// §3.8b/§3.10.2 — declare one editable value, at Setup. Registration is the ONLY
// thing that makes a value writable; publication, browsability and DATA_WRITE
// never are. All inputs are explicit for TwinCAT 4024 compatibility.
//
// A duplicate key is refused and the FIRST registration stands, because nothing
// here can tell which of the two the author meant. The refusal travels back
// through Setup, where a composition root sees it — rather than an operator
// discovering it later at a control that writes the wrong field.
METHOD M_RegisterConfigWrite : BOOL
VAR_INPUT
    Key           : STRING(160);
    Item          : STRING(255);
    Revision      : UDINT;
    Kind          : E_ConfigKind;
    ValueType     : E_ConfigValueType;
    Storage       : E_ConfigStorage;
    pTarget       : PVOID;
    RequiresReady : BOOL;
    HasMinimum    : BOOL;
    HasMaximum    : BOOL;
    Minimum       : LREAL;
    Maximum       : LREAL;
    Unit          : E_EngUnit;     // NONE = no unit; the HMI shows none
    LabelKey      : STRING(160);
    MaxLength     : UINT;
    EnumDomain    : STRING(255);
    EnumLabelKey  : STRING(80);    // '' = the values are shown as they are
END_VAR
VAR
    i : INT;
END_VAR
M_RegisterConfigWrite := FALSE;
IF _pConfigWrite = 0 THEN _pConfigWrite := ADR(_configWrite); END_IF
IF (Key = '') OR (Revision = 0) OR (pTarget = 0)
OR (Storage = E_ConfigStorage.NONE)
OR (_nConfigWrite >= _configCapacity) THEN
    RETURN;
END_IF
// A text target has a size this code cannot see. Storing 80 characters
// into a STRING(16) would corrupt whatever follows it, so the capacity is
// declared here and the store never exceeds it.
IF (Storage = E_ConfigStorage.AS_STRING)
AND ((MaxLength = 0) OR (MaxLength > 80)) THEN
    RETURN;
END_IF
IF HasMinimum AND HasMaximum AND (Minimum > Maximum) THEN
    RETURN;                                  // an empty range accepts nothing
END_IF
// §3.8e - a line value, and only a line value, is keyed 'line.'. A root publishes
// the line it references under its OWN scope, so the prefix is what keeps the
// line's keys and the root's apart; a mismatch in either direction fails closed.
IF (Kind = E_ConfigKind.LINE_CFG) <> (LEFT(Key, 5) = 'line.') THEN
    RETURN;
END_IF
FOR i := 1 TO _nConfigWrite DO
    IF _pConfigWrite[i - 1].Key = Key THEN
        RETURN;                              // duplicate (Scope, WriteKey): fail closed
    END_IF
END_FOR
_nConfigWrite := _nConfigWrite + 1;
_pConfigWrite[_nConfigWrite - 1].Key := Key;
_pConfigWrite[_nConfigWrite - 1].Item := Item;
_pConfigWrite[_nConfigWrite - 1].Revision := Revision;
_pConfigWrite[_nConfigWrite - 1].Kind := Kind;
_pConfigWrite[_nConfigWrite - 1].ValueType := ValueType;
_pConfigWrite[_nConfigWrite - 1].Storage := Storage;
_pConfigWrite[_nConfigWrite - 1].pTarget := pTarget;
_pConfigWrite[_nConfigWrite - 1].RequiresReady := RequiresReady;
_pConfigWrite[_nConfigWrite - 1].HasMinimum := HasMinimum;
_pConfigWrite[_nConfigWrite - 1].HasMaximum := HasMaximum;
_pConfigWrite[_nConfigWrite - 1].Minimum := Minimum;
_pConfigWrite[_nConfigWrite - 1].Maximum := Maximum;
_pConfigWrite[_nConfigWrite - 1].Unit := Unit;
_pConfigWrite[_nConfigWrite - 1].LabelKey := LabelKey;
_pConfigWrite[_nConfigWrite - 1].MaxLength := MaxLength;
_pConfigWrite[_nConfigWrite - 1].EnumDomain := EnumDomain;
_pConfigWrite[_nConfigWrite - 1].EnumLabelKey := EnumLabelKey;
M_RegisterConfigWrite := TRUE;
END_METHOD

// §3.8c - offer a capture for an ALREADY-REGISTERED editable value. Called at
// Setup, after the M_RegisterConfigWrite that declares the field.
//
// Refused when the key is not registered, which is §3.8c(a) enforced where it
// cannot be bypassed: capture changes how the number arrives, never which
// numbers may change. pSource shall point at a value the module already
// publishes (§3.8c(b)) - the operator has to be able to see the number that is
// about to be stored, on the same screen, before storing it.
METHOD M_RegisterCapture : BOOL
VAR_INPUT
    WriteKey       : STRING(160);
    pSource        : PVOID;
    SourceStorage  : E_ConfigStorage;
END_VAR
VAR
    i : INT;
END_VAR
M_RegisterCapture := FALSE;
IF (WriteKey = '') OR (pSource = 0) OR (SourceStorage = E_ConfigStorage.NONE) THEN
    RETURN;
END_IF
FOR i := 1 TO _nConfigWrite DO
    IF _pConfigWrite[i - 1].Key = WriteKey THEN
        _pConfigWrite[i - 1].pCapture       := pSource;
        _pConfigWrite[i - 1].CaptureStorage := SourceStorage;
        M_RegisterCapture := TRUE;
        RETURN;
    END_IF
END_FOR
END_METHOD

// §3.8c - read the live source as text, so the capture rejoins the ordinary
// write path instead of growing a second typed store. One conversion, one
// validator, one storage routine.
METHOD PRIVATE _M_ReadCaptureText : STRING(255)
VAR_INPUT
    Idx : INT;
END_VAR
VAR
    pB : POINTER TO BOOL;
    pI : POINTER TO INT;
    pD : POINTER TO DINT;
    pU : POINTER TO UDINT;
    pR : POINTER TO REAL;
    pL : POINTER TO LREAL;
    pT : POINTER TO TIME;
    pS : POINTER TO STRING(80);
END_VAR
_M_ReadCaptureText := '';
CASE _pConfigWrite[Idx - 1].CaptureStorage OF
    E_ConfigStorage.AS_BOOL:
        pB := _pConfigWrite[Idx - 1].pCapture;
        _M_ReadCaptureText := SEL(pB^, 'FALSE', 'TRUE');
    E_ConfigStorage.AS_INT:
        pI := _pConfigWrite[Idx - 1].pCapture;
        _M_ReadCaptureText := INT_TO_STRING(pI^);
    E_ConfigStorage.AS_DINT:
        pD := _pConfigWrite[Idx - 1].pCapture;
        _M_ReadCaptureText := DINT_TO_STRING(pD^);
    E_ConfigStorage.AS_UDINT:
        pU := _pConfigWrite[Idx - 1].pCapture;
        _M_ReadCaptureText := UDINT_TO_STRING(pU^);
    E_ConfigStorage.AS_REAL:
        pR := _pConfigWrite[Idx - 1].pCapture;
        _M_ReadCaptureText := REAL_TO_STRING(pR^);
    E_ConfigStorage.AS_LREAL:
        pL := _pConfigWrite[Idx - 1].pCapture;
        _M_ReadCaptureText := LREAL_TO_STRING(pL^);
    E_ConfigStorage.AS_TIME:
        // Whole milliseconds, per the HMI number contract (§3.8b).
        pT := _pConfigWrite[Idx - 1].pCapture;
        _M_ReadCaptureText := DWORD_TO_STRING(TIME_TO_DWORD(pT^));
    E_ConfigStorage.AS_STRING:
        pS := _pConfigWrite[Idx - 1].pCapture;
        _M_ReadCaptureText := pS^;
ELSE
    // Defined ELSE (S5.6): an unset or unknown source class yields empty text,
    // which the write path then refuses to parse. Fail-closed - a capture that
    // cannot read its source stores nothing rather than storing a zero.
    _M_ReadCaptureText := '';
END_CASE
END_METHOD

// §3.8d - put an already-registered value into a data class, and/or raise
// its own minimum levels. Public on purpose: a module TYPE may call it at Setup,
// and so may a composition root that wants a library value in one of the
// PROJECT's classes (a library cannot know a project's classes). The minimums
// only ever raise the class level - see FB_AccessManager.M_DataLevel.
METHOD M_SetConfigAccess : BOOL
VAR_INPUT
    WriteKey      : STRING(160);
    ClassId       : STRING(80);
    MinReadLevel  : E_AccessLevel;
    MinWriteLevel : E_AccessLevel;
END_VAR
VAR
    i : INT;
END_VAR
M_SetConfigAccess := FALSE;
IF (WriteKey = '') OR (LEN(ClassId) > 40)
OR (TO_DINT(MinReadLevel) < TO_DINT(E_AccessLevel.NONE))
OR (TO_DINT(MinReadLevel) > TO_DINT(E_AccessLevel.ADMIN))
OR (TO_DINT(MinWriteLevel) < TO_DINT(E_AccessLevel.NONE))
OR (TO_DINT(MinWriteLevel) > TO_DINT(E_AccessLevel.ADMIN)) THEN
    RETURN;
END_IF
FOR i := 1 TO _nConfigWrite DO
    IF _pConfigWrite[i - 1].Key = WriteKey THEN
        _pConfigWrite[i - 1].ClassId := ClassId;
        _pConfigWrite[i - 1].MinReadLevel := MinReadLevel;
        _pConfigWrite[i - 1].MinWriteLevel := MinWriteLevel;
        M_SetConfigAccess := TRUE;
        RETURN;
    END_IF
END_FOR
END_METHOD

// §3.8d I_ConfigSource - this module's own registry only; composites recurse.
METHOD M_ConfigAccessOf : BOOL
VAR_INPUT
    Scope    : STRING(255);
    WriteKey : STRING(160);
END_VAR
VAR_IN_OUT
    Grant : ST_ConfigAccess;
END_VAR
VAR
    i : INT;
END_VAR
M_ConfigAccessOf := FALSE;
IF (WriteKey = '') OR (Scope <> Status.Name) THEN
    RETURN;
END_IF
FOR i := 1 TO _nConfigWrite DO
    IF _pConfigWrite[i - 1].Key = WriteKey THEN
        Grant.Kind := _pConfigWrite[i - 1].Kind;
        Grant.ClassId := _pConfigWrite[i - 1].ClassId;
        Grant.MinReadLevel := _pConfigWrite[i - 1].MinReadLevel;
        Grant.MinWriteLevel := _pConfigWrite[i - 1].MinWriteLevel;
        M_ConfigAccessOf := TRUE;
        RETURN;
    END_IF
END_FOR
END_METHOD

// §3.8e - TRUE while this module's registered values may not be changed by a
// client: still published, as Writable := FALSE, and refused by the write and
// staging paths. The base is always writable; a line-data MIRROR is not.
METHOD PROTECTED _M_ConfigReadOnly : BOOL
_M_ConfigReadOnly := FALSE;
END_METHOD

// §3.8b — a numeric editable value. Bounds are mandatory here on purpose: an
// unbounded number is the one a client can set to anything, and "what is the
// valid range" is a question the owning module is the only one able to answer.
// Use M_RegisterConfigWrite directly for an unbounded or higher-revision value.
METHOD M_RegisterConfigNumber : BOOL
VAR_INPUT
    Key           : STRING(160);
    Item          : STRING(255);
    LabelKey      : STRING(160);
    Unit          : E_EngUnit;     // every number declares one; NONE = unitless
    Kind          : E_ConfigKind;
    Storage       : E_ConfigStorage;
    pTarget       : PVOID;
    Minimum       : LREAL;
    Maximum       : LREAL;
    RequiresReady : BOOL;
END_VAR
M_RegisterConfigNumber := M_RegisterConfigWrite(Key := Key, Item := Item,
    Revision := 1, Kind := Kind, ValueType := E_ConfigValueType.NUMBER,
    Storage := Storage, pTarget := pTarget, RequiresReady := RequiresReady,
    HasMinimum := TRUE, HasMaximum := TRUE, Minimum := Minimum, Maximum := Maximum,
    Unit := Unit, LabelKey := LabelKey, MaxLength := 0, EnumDomain := '',
    EnumLabelKey := '');
END_METHOD

// §3.8b — an editable TIME, carried and edited as whole milliseconds (the HMI
// validates DURATION as a number; TC3 §3.8 explains the enum spelling).
METHOD M_RegisterConfigDuration : BOOL
VAR_INPUT
    Key           : STRING(160);
    Item          : STRING(255);
    LabelKey      : STRING(160);
    Kind          : E_ConfigKind;
    pTarget       : POINTER TO TIME;
    MinimumMs     : UDINT;
    MaximumMs     : UDINT;
    RequiresReady : BOOL;
END_VAR
M_RegisterConfigDuration := M_RegisterConfigWrite(Key := Key, Item := Item,
    Revision := 1, Kind := Kind, ValueType := E_ConfigValueType.DURATION,
    Storage := E_ConfigStorage.AS_TIME, pTarget := pTarget,
    RequiresReady := RequiresReady, HasMinimum := TRUE, HasMaximum := TRUE,
    Minimum := TO_LREAL(MinimumMs), Maximum := TO_LREAL(MaximumMs),
    Unit := E_EngUnit.MILLISECOND, LabelKey := LabelKey, MaxLength := 0,
    EnumDomain := '', EnumLabelKey := '');
END_METHOD

// §3.8b — an editable BOOL. The exact domain is declared so a client renders a
// choice rather than a free-text field, and so 'yes' is rejected rather than
// silently read as FALSE.
METHOD M_RegisterConfigFlag : BOOL
VAR_INPUT
    Key           : STRING(160);
    Item          : STRING(255);
    LabelKey      : STRING(160);
    Kind          : E_ConfigKind;
    pTarget       : POINTER TO BOOL;
    RequiresReady : BOOL;
END_VAR
M_RegisterConfigFlag := M_RegisterConfigWrite(Key := Key, Item := Item,
    Revision := 1, Kind := Kind, ValueType := E_ConfigValueType.BOOLEAN,
    Storage := E_ConfigStorage.AS_BOOL, pTarget := pTarget,
    RequiresReady := RequiresReady, HasMinimum := FALSE, HasMaximum := FALSE,
    Minimum := 0.0, Maximum := 0.0, Unit := E_EngUnit.NONE, LabelKey := LabelKey,
    MaxLength := 0, EnumDomain := 'TRUE|FALSE', EnumLabelKey := '');
END_METHOD

// §3.8b/§3.10.2 - an editable value that is one of a fixed set, e.g. an
// enumeration stored as its ordinal. Domain lists the exact accepted values
// ('0|1|2'); EnumLabelKey is the catalog prefix the HMI labels each one with
// ('<EnumLabelKey>.<value>'), so a client renders a translated choice and
// anything outside the domain is refused, never read as a default.
METHOD M_RegisterConfigChoice : BOOL
VAR_INPUT
    Key           : STRING(160);
    Item          : STRING(255);
    LabelKey      : STRING(160);
    Kind          : E_ConfigKind;
    Storage       : E_ConfigStorage;
    pTarget       : PVOID;
    Domain        : STRING(255);
    EnumLabelKey  : STRING(80);
    RequiresReady : BOOL;
END_VAR
M_RegisterConfigChoice := FALSE;
IF Domain = '' THEN
    RETURN;                                  // a choice with no choices accepts nothing
END_IF
M_RegisterConfigChoice := M_RegisterConfigWrite(Key := Key, Item := Item,
    Revision := 1, Kind := Kind, ValueType := E_ConfigValueType.NUMBER,
    Storage := Storage, pTarget := pTarget, RequiresReady := RequiresReady,
    HasMinimum := FALSE, HasMaximum := FALSE, Minimum := 0.0, Maximum := 0.0,
    Unit := E_EngUnit.NONE, LabelKey := LabelKey, MaxLength := 0,
    EnumDomain := Domain, EnumLabelKey := EnumLabelKey);
END_METHOD

// §3.8b/§3.10.2 I_ConfigSource — apply one registered write to THIS module.
// The root has already checked DATA_WRITE and subtree ownership; what is left is
// everything only the owner knows. Scope selects the module, so the recursive
// walk asks each module in turn and exactly the one that registered the key
// answers TRUE. An unknown key, a stale revision, or a value the module refuses
// all return FALSE and change nothing.
METHOD M_ApplyConfigWrite : BOOL
VAR_INPUT
    Scope     : STRING(255);
    WriteKey  : STRING(160);
    Revision  : UDINT;
    TextValue : STRING(255);
    RootReady : BOOL;
END_VAR
VAR
    i : INT;
END_VAR
M_ApplyConfigWrite := FALSE;
IF (WriteKey = '') OR (Scope <> Status.Name) OR _M_ConfigReadOnly() THEN
    RETURN;
END_IF
FOR i := 1 TO _nConfigWrite DO
    IF _pConfigWrite[i - 1].Key = WriteKey THEN
        IF _pConfigWrite[i - 1].Revision <> Revision THEN
            RETURN;              // stale capability — the client's metadata is old
        END_IF
        IF _pConfigWrite[i - 1].RequiresReady AND NOT RootReady THEN
            RETURN;
        END_IF
        // The type-specific hook sees the candidate BEFORE anything is stored, so
        // a refusal here is indistinguishable from a range refusal: nothing moved.
        IF NOT _M_OnConfigWrite(WriteKey := WriteKey, TextValue := TextValue) THEN
            RETURN;
        END_IF
        M_ApplyConfigWrite := _M_StoreConfigValue(Idx := i, TextValue := TextValue,
            Commit := TRUE);
        RETURN;
    END_IF
END_FOR
END_METHOD

// §3.8c - apply a capture to THIS module. Resolves the live value and then hands
// it to the ordinary write path, so validation, the type's own invariants, range,
// domain and storage are the SAME code a typed write goes through. A machine-
// supplied number is not more trustworthy than a human-supplied one (§14).
METHOD M_ApplyCapture : BOOL
VAR_INPUT
    Scope     : STRING(255);
    WriteKey  : STRING(160);
    Revision  : UDINT;
    RootReady : BOOL;
END_VAR
VAR
    i : INT;
END_VAR
M_ApplyCapture := FALSE;
IF (WriteKey = '') OR (Scope <> Status.Name) THEN
    RETURN;
END_IF
FOR i := 1 TO _nConfigWrite DO
    IF _pConfigWrite[i - 1].Key = WriteKey THEN
        // No capture registered for this field: refuse rather than fall back to
        // some default, so an unoffered capture can never quietly store a zero.
        IF _pConfigWrite[i - 1].pCapture = 0 THEN
            RETURN;
        END_IF
        M_ApplyCapture := M_ApplyConfigWrite(Scope := Scope, WriteKey := WriteKey,
            Revision := Revision, TextValue := _M_ReadCaptureText(Idx := i),
            RootReady := RootReady);
        RETURN;
    END_IF
END_FOR
END_METHOD

// §3.10.2 — module-specific invariants a generic type/range check cannot state:
// a value that must stay below another, a device that must be idle first. The
// base accepts; the framework still validates revision, type, range and domain
// and stores only after this returns TRUE. Two rules for an override: it shall
// have no side effects, because this runs on a candidate that may still be
// rejected; and it sees the RAW text, not a parsed value — 'abc' reaches it
// exactly as '7' does, so it must never assume the candidate is a number.
METHOD PROTECTED _M_OnConfigWrite : BOOL
VAR_INPUT
    WriteKey  : STRING(160);
    TextValue : STRING(255);
END_VAR
_M_OnConfigWrite := TRUE;
END_METHOD

// §3.8b/§5.6 — validate a candidate completely, then store it. Every rejection
// happens before the first byte moves, so a refused write leaves the module
// exactly as it was. Range is checked against BOTH the declared bounds and the
// storage type's own limits: a DINT field with no declared maximum still cannot
// be handed 1E30.
//
// Commit := FALSE runs the IDENTICAL validation and stores nothing. That is the
// staging pass of a §3.8b set load, and it deliberately shares this code rather
// than restating the rules: a validator that can disagree with the writer is
// worse than no validator, because it makes an all-or-nothing load claim an
// atomicity it does not have.
METHOD PROTECTED _M_StoreConfigValue : BOOL
VAR_INPUT
    Idx       : INT;
    TextValue : STRING(255);
    Commit    : BOOL;
END_VAR
VAR
    num : LREAL;
    pB  : POINTER TO BOOL;
    pI  : POINTER TO INT;
    pD  : POINTER TO DINT;
    pU  : POINTER TO UDINT;
    pR  : POINTER TO REAL;
    pL  : POINTER TO LREAL;
    pT  : POINTER TO TIME;
    pS  : POINTER TO STRING(80);
END_VAR
_M_StoreConfigValue := FALSE;
IF (Idx < 1) OR (Idx > _nConfigWrite) OR (_pConfigWrite[Idx - 1].pTarget = 0) THEN
    RETURN;
END_IF
// A declared domain is exact and is checked on the raw text, whatever the type.
IF _pConfigWrite[Idx - 1].EnumDomain <> '' THEN
    IF NOT _M_InEnumDomain(Domain := _pConfigWrite[Idx - 1].EnumDomain,
            Text := TextValue) THEN
        RETURN;
    END_IF
END_IF
IF _pConfigWrite[Idx - 1].Storage = E_ConfigStorage.AS_BOOL THEN
    pB := _M_Target(Idx := Idx);
    IF (TextValue = 'TRUE') OR (TextValue = 'true') OR (TextValue = 'True')
    OR (TextValue = '1') THEN
        IF Commit THEN
            pB^ := TRUE;
        END_IF
    ELSIF (TextValue = 'FALSE') OR (TextValue = 'false') OR (TextValue = 'False')
    OR (TextValue = '0') THEN
        IF Commit THEN
            pB^ := FALSE;
        END_IF
    ELSE
        RETURN;
    END_IF
    _M_StoreConfigValue := TRUE;
    RETURN;
END_IF
IF _pConfigWrite[Idx - 1].Storage = E_ConfigStorage.AS_STRING THEN
    IF TO_UINT(LEN(TextValue)) > _pConfigWrite[Idx - 1].MaxLength THEN
        RETURN;                              // would truncate: reject, never trim
    END_IF
    IF Commit THEN
        pS := _M_Target(Idx := Idx);
        pS^ := TextValue;
    END_IF
    _M_StoreConfigValue := TRUE;
    RETURN;
END_IF
// Everything else is numeric.
IF NOT F_TryParseNumber(Text := TextValue, Value => num) THEN
    RETURN;
END_IF
IF _pConfigWrite[Idx - 1].HasMinimum AND (num < _pConfigWrite[Idx - 1].Minimum) THEN
    RETURN;
END_IF
IF _pConfigWrite[Idx - 1].HasMaximum AND (num > _pConfigWrite[Idx - 1].Maximum) THEN
    RETURN;
END_IF
CASE _pConfigWrite[Idx - 1].Storage OF
    E_ConfigStorage.AS_INT:
        IF (num < -32768.0) OR (num > 32767.0) THEN
            RETURN;
        END_IF
        // Two statements, not one condition: IEC 61131-3 does not mandate
        // short-circuit evaluation and TwinCAT's option for it is off by
        // default, so a combined test would still convert a value the range
        // check is there to reject (§5.6).
        IF num <> TO_LREAL(TO_LINT(num)) THEN
            RETURN;
        END_IF
        IF Commit THEN
            pI := _M_Target(Idx := Idx);
            pI^ := LREAL_TO_INT(num);
        END_IF
    E_ConfigStorage.AS_DINT:
        IF (num < -2147483648.0) OR (num > 2147483647.0) THEN
            RETURN;
        END_IF
        IF num <> TO_LREAL(TO_LINT(num)) THEN
            RETURN;
        END_IF
        IF Commit THEN
            pD := _M_Target(Idx := Idx);
            pD^ := LREAL_TO_DINT(num);
        END_IF
    E_ConfigStorage.AS_UDINT:
        IF (num < 0.0) OR (num > 4294967295.0) THEN
            RETURN;
        END_IF
        IF num <> TO_LREAL(TO_LINT(num)) THEN
            RETURN;
        END_IF
        IF Commit THEN
            pU := _M_Target(Idx := Idx);
            pU^ := LREAL_TO_UDINT(num);
        END_IF
    E_ConfigStorage.AS_REAL:
        IF (num < -3.402823E38) OR (num > 3.402823E38) THEN
            RETURN;
        END_IF
        IF Commit THEN
            pR := _M_Target(Idx := Idx);
            pR^ := LREAL_TO_REAL(num);
        END_IF
    E_ConfigStorage.AS_LREAL:
        IF Commit THEN
            pL := _M_Target(Idx := Idx);
            pL^ := num;
        END_IF
    E_ConfigStorage.AS_TIME:
        // Whole milliseconds: a duration is not a place for a rounding surprise.
        IF (num < 0.0) OR (num > 4294967295.0) THEN
            RETURN;
        END_IF
        IF num <> TO_LREAL(TO_LINT(num)) THEN
            RETURN;
        END_IF
        IF Commit THEN
            pT := _M_Target(Idx := Idx);
            pT^ := UDINT_TO_TIME(LREAL_TO_UDINT(num));
        END_IF
ELSE
    RETURN;
END_CASE
_M_StoreConfigValue := TRUE;
END_METHOD

// §3.10.2 — the current value of a registered entry, in the serialization the
// client validates and writes back. Read live from the target every walk: a
// cached copy would let the manifest disagree with the machine.
METHOD PROTECTED _M_ConfigValueText : STRING(255)
VAR_INPUT
    Idx : INT;
END_VAR
VAR
    pB : POINTER TO BOOL;
    pI : POINTER TO INT;
    pD : POINTER TO DINT;
    pU : POINTER TO UDINT;
    pR : POINTER TO REAL;
    pL : POINTER TO LREAL;
    pT : POINTER TO TIME;
    pS : POINTER TO STRING(80);
END_VAR
_M_ConfigValueText := '';
IF (Idx < 1) OR (Idx > _nConfigWrite) OR (_pConfigWrite[Idx - 1].pTarget = 0) THEN
    RETURN;
END_IF
CASE _pConfigWrite[Idx - 1].Storage OF
    E_ConfigStorage.AS_BOOL:
        pB := _M_Target(Idx := Idx);
        IF pB^ THEN
            _M_ConfigValueText := 'TRUE';
        ELSE
            _M_ConfigValueText := 'FALSE';
        END_IF
    E_ConfigStorage.AS_INT:
        pI := _M_Target(Idx := Idx);
        _M_ConfigValueText := TO_STRING(pI^);
    E_ConfigStorage.AS_DINT:
        pD := _M_Target(Idx := Idx);
        _M_ConfigValueText := TO_STRING(pD^);
    E_ConfigStorage.AS_UDINT:
        pU := _M_Target(Idx := Idx);
        _M_ConfigValueText := TO_STRING(pU^);
    E_ConfigStorage.AS_REAL:
        pR := _M_Target(Idx := Idx);
        _M_ConfigValueText := TO_STRING(pR^);
    E_ConfigStorage.AS_LREAL:
        pL := _M_Target(Idx := Idx);
        _M_ConfigValueText := TO_STRING(pL^);
    E_ConfigStorage.AS_TIME:
        pT := _M_Target(Idx := Idx);
        _M_ConfigValueText := TO_STRING(TIME_TO_UDINT(pT^));
    E_ConfigStorage.AS_STRING:
        pS := _M_Target(Idx := Idx);
        _M_ConfigValueText := pS^;
END_CASE
END_METHOD

// §3.10.2 — exact membership in a pipe-separated domain. Exact means exact: no
// trimming, no case folding. The client was given this list and can send one of
// its entries.
METHOD PRIVATE _M_InEnumDomain : BOOL
VAR_INPUT
    Domain : STRING(255);
    Text   : STRING(255);
END_VAR
VAR
    rest  : STRING(255);
    token : STRING(255);
    pos   : INT;
    i     : INT;
END_VAR
_M_InEnumDomain := FALSE;
rest := Domain;
FOR i := 1 TO 32 DO                          // bounded scan (§5.6)
    IF rest = '' THEN
        RETURN;
    END_IF
    pos := FIND(rest, '|');
    IF pos = 0 THEN
        token := rest;
        rest := '';
    ELSE
        token := LEFT(rest, pos - 1);
        rest := MID(rest, TO_INT(LEN(rest)) - pos, pos + 1);
    END_IF
    IF token = Text THEN
        _M_InEnumDomain := TRUE;
        RETURN;
    END_IF
END_FOR
END_METHOD

// §3.8b I_ConfigSource — would this write be accepted? Byte-for-byte the
// lookup and gating of M_ApplyConfigWrite, then the shared validator with
// Commit := FALSE. Nothing in this module changes, including through the
// type-specific invariant hook, which §3.10.2 already requires to be free of
// side effects because it runs on a candidate that may still be rejected.
METHOD M_StageConfigWrite : BOOL
VAR_INPUT
    Scope     : STRING(255);
    WriteKey  : STRING(160);
    Revision  : UDINT;
    TextValue : STRING(255);
    RootReady : BOOL;
END_VAR
VAR
    i : INT;
END_VAR
M_StageConfigWrite := FALSE;
IF (WriteKey = '') OR (Scope <> Status.Name) OR _M_ConfigReadOnly() THEN
    RETURN;
END_IF
FOR i := 1 TO _nConfigWrite DO
    IF _pConfigWrite[i - 1].Key = WriteKey THEN
        IF _pConfigWrite[i - 1].Revision <> Revision THEN
            RETURN;
        END_IF
        IF _pConfigWrite[i - 1].RequiresReady AND NOT RootReady THEN
            RETURN;
        END_IF
        IF NOT _M_OnConfigWrite(WriteKey := WriteKey, TextValue := TextValue) THEN
            RETURN;
        END_IF
        M_StageConfigWrite := _M_StoreConfigValue(Idx := i, TextValue := TextValue,
            Commit := FALSE);
        RETURN;
    END_IF
END_FOR
END_METHOD

// §3.8b — the restore rule for one retained StationCfg image, written ONCE here
// so no module type carries its own copy of it (§1.1 O1).
//
// Every StationCfg structure shall carry SchemaVersion : UINT as its FIRST
// member, and this decides what a given value of it means:
//
//   version = SchemaVersion  -> restored. Returns TRUE; the caller keeps the
//                               retained values and does nothing.
//   version = 0              -> never written. A first boot has lost nothing,
//                               so it initializes SILENTLY: returns FALSE with
//                               no annunciation, and the caller writes defaults.
//   anything else            -> a REAL image was rejected. Returns FALSE and
//                               records the loss for the root to annunciate with
//                               this module's canonical path.
//
// The version is stamped forward either way, so the next boot is an ordinary
// restore rather than a repeated annunciation. What is NOT done is reading the
// unrecognized image by field position: that is precisely how a changed layout
// becomes a plausible wrong number instead of an honest default.
//
// The consequence of a loss belongs to the deployment, not to this module —
// E_ConfigRestorePolicy at the root decides whether the station runs and
// annunciates or refuses START_STOP until an ENGINEER acknowledges. A module
// that faulted itself here would take that decision away from the deployment.
METHOD M_RestoreStationCfg : BOOL
VAR_INPUT
    pVersion      : POINTER TO UINT;   // ADR of the structure's FIRST member
    SchemaVersion : UINT;              // the layout this build understands
END_VAR
M_RestoreStationCfg := FALSE;
IF pVersion = 0 THEN
    RETURN;                              // unwired: defaults, and never a claim
END_IF
IF SchemaVersion = 0 THEN
    RETURN;                              // 0 is reserved for "never written"
END_IF
IF pVersion^ = SchemaVersion THEN
    M_RestoreStationCfg := TRUE;
    RETURN;
END_IF
IF pVersion^ <> 0 THEN
    // A real image was rejected. The station will run on defaults and it will
    // say so — the difference between an empty machine and one that has just
    // lost its commissioning is exactly what an operator needs told.
    _restoreLost := TRUE;
    _restoreFound := pVersion^;
    _restoreExpected := SchemaVersion;
END_IF
pVersion^ := SchemaVersion;
END_METHOD

// §3.8b I_ConfigSource — hand the root this module's unreported restore loss,
// exactly once. Taking it clears the slot, so the root can drain the whole
// subtree in a loop and each loss is annunciated one time per boot.
METHOD M_TakeRestoreLoss : BOOL
VAR_OUTPUT
    Path     : STRING(80);
    Expected : UINT;
    Found    : UINT;
END_VAR
M_TakeRestoreLoss := FALSE;
Path := '';
Expected := 0;
Found := 0;
IF NOT _restoreLost THEN
    RETURN;
END_IF
_restoreLost := FALSE;
Path := Status.Name;
Expected := _restoreExpected;
Found := _restoreFound;
M_TakeRestoreLoss := TRUE;
END_METHOD

// §7.6.1 I_ManualTarget - answer for THIS module only. Same shape as
// M_ApplyConfigWrite: the walk asks every module and exactly the one whose
// Scope matches replies, so routing is a property of registration rather than
// of a chain somebody maintains by hand.
METHOD M_ApplyManual : BOOL
VAR_INPUT
    Scope : STRING(255);
    Value : DINT;
END_VAR
M_ApplyManual := FALSE;
IF Scope <> Status.Name THEN
    RETURN;
END_IF
// ManualCommand still validates the value against the published catalogue and
// still runs the §6.1 lifecycle. Reaching the module is all this adds.
M_ApplyManual := ManualCommand(Value := Value);
END_METHOD

// §7.6.1a I_ManualTarget - the held-command twin of M_ApplyManual. A type with
// no held commands inherits RequestHeldCommand's refusal, so an unsupported
// hold is a defined FALSE.
METHOD M_ApplyHeld : BOOL
VAR_INPUT
    Scope  : STRING(255);
    Value  : DINT;
    Enable : ST_ManualEnableStatus;
END_VAR
M_ApplyHeld := FALSE;
IF Scope <> Status.Name THEN
    RETURN;
END_IF
M_ApplyHeld := RequestHeldCommand(Value := Value, Enable := Enable);
END_METHOD

// Optional owner storage selected before any registration; base modules keep twelve slots.
METHOD PROTECTED _M_UseConfigRegistry : BOOL
VAR_INPUT
    pRecords : POINTER TO ST_ConfigWriteDef;
    Capacity : INT;
END_VAR
_M_UseConfigRegistry := FALSE;
IF (_nConfigWrite <> 0) OR (pRecords = 0) OR (Capacity < 1)
OR (Capacity > PL_Fraktal.MAX_LINE_RECORDS) THEN RETURN; END_IF
_pConfigWrite := pRecords;
_configCapacity := Capacity;
_M_UseConfigRegistry := TRUE;
END_METHOD

END_FUNCTION_BLOCK

// ---- Platform/F_RationalizeDiagnostic.TcPOU
// Core §8.9 — apply the one generated priority/category to a diagnostic at its
// source. Unknown external reasons keep the caller values until their owning
// AlarmLog joins a validated runtime record.
FUNCTION F_RationalizeDiagnostic : BOOL
VAR_IN_OUT
    Diag : ST_Diagnostic;
END_VAR
VAR
    meta : ST_AlarmMeta;
END_VAR

F_RationalizeDiagnostic := F_ReasonMeta(
    Reason := Diag.ReasonCode, Meta := meta);
IF F_RationalizeDiagnostic THEN
    Diag.Severity := meta.Priority;
    Diag.Category := meta.Category;
END_IF

END_FUNCTION

// ---- Platform/F_ReasonMeta.TcPOU
// Core §8.9 — resolve one generated rationalization by ReasonCode.
FUNCTION F_ReasonMeta : BOOL
VAR_INPUT
    Reason : E_Reason;
END_VAR
VAR_IN_OUT
    Meta : ST_AlarmMeta;
END_VAR
VAR
    i : INT;
    candidate : ST_AlarmMeta;
END_VAR

F_ReasonMeta := FALSE;
FOR i := 1 TO PL_ReasonCatalog.COUNT DO
    IF F_ReasonMetaByIndex(Index := i, Meta := candidate)
    AND (candidate.ReasonCode = Reason) THEN
        Meta := candidate;
        F_ReasonMeta := TRUE;
        RETURN;
    END_IF
END_FOR

END_FUNCTION

// ---- Platform/F_ReasonMetaByIndex.TcPOU
// GENERATED FILE — DO NOT EDIT. Core §8.8/§8.9 complete catalog projection.
FUNCTION F_ReasonMetaByIndex : BOOL
VAR_INPUT
    Index : INT;
END_VAR
VAR_IN_OUT
    Meta : ST_AlarmMeta;
END_VAR

F_ReasonMetaByIndex := FALSE;
Meta.ReasonCode := E_Reason.NONE;
Meta.OperatorAction := '';
Meta.Consequence := '';
Meta.Priority := E_Severity.LOW;
Meta.Category := E_Category.PROCESS;
Meta.Shelvable := FALSE;
CASE Index OF
    1:
        Meta.ReasonCode := 10;
        Meta.OperatorAction := 'std.reason.10.action';
        Meta.Consequence := 'std.reason.10.consequence';
        Meta.Priority := E_Severity.MED;
        Meta.Category := E_Category.SYSTEM;
        Meta.Shelvable := FALSE;
    2:
        Meta.ReasonCode := 11;
        Meta.OperatorAction := 'std.reason.11.action';
        Meta.Consequence := 'std.reason.11.consequence';
        Meta.Priority := E_Severity.LOW;
        Meta.Category := E_Category.SYSTEM;
        Meta.Shelvable := TRUE;
    3:
        Meta.ReasonCode := 12;
        Meta.OperatorAction := 'std.reason.12.action';
        Meta.Consequence := 'std.reason.12.consequence';
        Meta.Priority := E_Severity.LOW;
        Meta.Category := E_Category.SYSTEM;
        Meta.Shelvable := TRUE;
    4:
        Meta.ReasonCode := 13;
        Meta.OperatorAction := 'std.reason.13.action';
        Meta.Consequence := 'std.reason.13.consequence';
        Meta.Priority := E_Severity.MED;
        Meta.Category := E_Category.SYSTEM;
        Meta.Shelvable := FALSE;
    5:
        Meta.ReasonCode := 14;
        Meta.OperatorAction := 'std.reason.14.action';
        Meta.Consequence := 'std.reason.14.consequence';
        Meta.Priority := E_Severity.MED;
        Meta.Category := E_Category.SYSTEM;
        Meta.Shelvable := FALSE;
    6:
        Meta.ReasonCode := 15;
        Meta.OperatorAction := 'std.reason.15.action';
        Meta.Consequence := 'std.reason.15.consequence';
        Meta.Priority := E_Severity.HIGH;
        Meta.Category := E_Category.SYSTEM;
        Meta.Shelvable := FALSE;
    7:
        Meta.ReasonCode := 16;
        Meta.OperatorAction := 'std.reason.16.action';
        Meta.Consequence := 'std.reason.16.consequence';
        Meta.Priority := E_Severity.LOW;
        Meta.Category := E_Category.SYSTEM;
        Meta.Shelvable := TRUE;
    8:
        Meta.ReasonCode := 17;
        Meta.OperatorAction := 'std.reason.17.action';
        Meta.Consequence := 'std.reason.17.consequence';
        Meta.Priority := E_Severity.LOW;
        Meta.Category := E_Category.SYSTEM;
        Meta.Shelvable := TRUE;
    9:
        Meta.ReasonCode := 18;
        Meta.OperatorAction := 'std.reason.18.action';
        Meta.Consequence := 'std.reason.18.consequence';
        Meta.Priority := E_Severity.MED;
        Meta.Category := E_Category.SYSTEM;
        Meta.Shelvable := FALSE;
    10:
        Meta.ReasonCode := 19;
        Meta.OperatorAction := 'std.reason.19.action';
        Meta.Consequence := 'std.reason.19.consequence';
        Meta.Priority := E_Severity.LOW;
        Meta.Category := E_Category.SYSTEM;
        Meta.Shelvable := TRUE;
    11:
        Meta.ReasonCode := 20;
        Meta.OperatorAction := 'std.reason.20.action';
        Meta.Consequence := 'std.reason.20.consequence';
        Meta.Priority := E_Severity.MED;
        Meta.Category := E_Category.SYSTEM;
        Meta.Shelvable := FALSE;
    12:
        Meta.ReasonCode := 21;
        Meta.OperatorAction := 'std.reason.21.action';
        Meta.Consequence := 'std.reason.21.consequence';
        Meta.Priority := E_Severity.LOW;
        Meta.Category := E_Category.SYSTEM;
        Meta.Shelvable := TRUE;
    13:
        Meta.ReasonCode := 2001;
        Meta.OperatorAction := 'std.reason.2001.action';
        Meta.Consequence := 'std.reason.2001.consequence';
        Meta.Priority := E_Severity.MED;
        Meta.Category := E_Category.PROCESS;
        Meta.Shelvable := FALSE;
    14:
        Meta.ReasonCode := 2002;
        Meta.OperatorAction := 'std.reason.2002.action';
        Meta.Consequence := 'std.reason.2002.consequence';
        Meta.Priority := E_Severity.LOW;
        Meta.Category := E_Category.PROCESS;
        Meta.Shelvable := FALSE;
    15:
        Meta.ReasonCode := 2003;
        Meta.OperatorAction := 'std.reason.2003.action';
        Meta.Consequence := 'std.reason.2003.consequence';
        Meta.Priority := E_Severity.MED;
        Meta.Category := E_Category.PROCESS;
        Meta.Shelvable := FALSE;
    16:
        Meta.ReasonCode := 2004;
        Meta.OperatorAction := 'std.reason.2004.action';
        Meta.Consequence := 'std.reason.2004.consequence';
        Meta.Priority := E_Severity.MED;
        Meta.Category := E_Category.PROCESS;
        Meta.Shelvable := FALSE;
    17:
        Meta.ReasonCode := 2005;
        Meta.OperatorAction := 'std.reason.2005.action';
        Meta.Consequence := 'std.reason.2005.consequence';
        Meta.Priority := E_Severity.LOW;
        Meta.Category := E_Category.PROCESS;
        Meta.Shelvable := TRUE;
    18:
        Meta.ReasonCode := 2006;
        Meta.OperatorAction := 'std.reason.2006.action';
        Meta.Consequence := 'std.reason.2006.consequence';
        Meta.Priority := E_Severity.MED;
        Meta.Category := E_Category.PROCESS;
        Meta.Shelvable := FALSE;
    19:
        Meta.ReasonCode := 2007;
        Meta.OperatorAction := 'std.reason.2007.action';
        Meta.Consequence := 'std.reason.2007.consequence';
        Meta.Priority := E_Severity.LOW;
        Meta.Category := E_Category.PROCESS;
        Meta.Shelvable := TRUE;
    20:
        Meta.ReasonCode := 2008;
        Meta.OperatorAction := 'std.reason.2008.action';
        Meta.Consequence := 'std.reason.2008.consequence';
        Meta.Priority := E_Severity.LOW;
        Meta.Category := E_Category.PROCESS;
        Meta.Shelvable := FALSE;
    21:
        Meta.ReasonCode := 2010;
        Meta.OperatorAction := 'std.reason.2010.action';
        Meta.Consequence := 'std.reason.2010.consequence';
        Meta.Priority := E_Severity.MED;
        Meta.Category := E_Category.SYSTEM;
        Meta.Shelvable := FALSE;
    22:
        Meta.ReasonCode := 2011;
        Meta.OperatorAction := 'std.reason.2011.action';
        Meta.Consequence := 'std.reason.2011.consequence';
        Meta.Priority := E_Severity.LOW;
        Meta.Category := E_Category.PROCESS;
        Meta.Shelvable := TRUE;
    23:
        Meta.ReasonCode := 2012;
        Meta.OperatorAction := 'std.reason.2012.action';
        Meta.Consequence := 'std.reason.2012.consequence';
        Meta.Priority := E_Severity.MED;
        Meta.Category := E_Category.SYSTEM;
        Meta.Shelvable := FALSE;
    24:
        Meta.ReasonCode := 2020;
        Meta.OperatorAction := 'std.reason.2020.action';
        Meta.Consequence := 'std.reason.2020.consequence';
        Meta.Priority := E_Severity.MED;
        Meta.Category := E_Category.SYSTEM;
        Meta.Shelvable := FALSE;
    25:
        Meta.ReasonCode := 2021;
        Meta.OperatorAction := 'std.reason.2021.action';
        Meta.Consequence := 'std.reason.2021.consequence';
        Meta.Priority := E_Severity.MED;
        Meta.Category := E_Category.SYSTEM;
        Meta.Shelvable := FALSE;
    26:
        Meta.ReasonCode := 2022;
        Meta.OperatorAction := 'std.reason.2022.action';
        Meta.Consequence := 'std.reason.2022.consequence';
        Meta.Priority := E_Severity.HIGH;
        Meta.Category := E_Category.PROCESS;
        Meta.Shelvable := FALSE;
    27:
        Meta.ReasonCode := 2023;
        Meta.OperatorAction := 'std.reason.2023.action';
        Meta.Consequence := 'std.reason.2023.consequence';
        Meta.Priority := E_Severity.MED;
        Meta.Category := E_Category.PROCESS;
        Meta.Shelvable := FALSE;
    28:
        Meta.ReasonCode := 2024;
        Meta.OperatorAction := '';
        Meta.Consequence := 'std.reason.2024.consequence';
        Meta.Priority := E_Severity.LOW;
        Meta.Category := E_Category.PROCESS;
        Meta.Shelvable := FALSE;
    29:
        Meta.ReasonCode := 2025;
        Meta.OperatorAction := '';
        Meta.Consequence := 'std.reason.2025.consequence';
        Meta.Priority := E_Severity.LOW;
        Meta.Category := E_Category.PROCESS;
        Meta.Shelvable := FALSE;
    30:
        Meta.ReasonCode := 2026;
        Meta.OperatorAction := '';
        Meta.Consequence := 'std.reason.2026.consequence';
        Meta.Priority := E_Severity.LOW;
        Meta.Category := E_Category.PROCESS;
        Meta.Shelvable := FALSE;
    31:
        Meta.ReasonCode := 2027;
        Meta.OperatorAction := '';
        Meta.Consequence := 'std.reason.2027.consequence';
        Meta.Priority := E_Severity.LOW;
        Meta.Category := E_Category.PROCESS;
        Meta.Shelvable := FALSE;
    32:
        Meta.ReasonCode := 2030;
        Meta.OperatorAction := 'std.reason.2030.action';
        Meta.Consequence := 'std.reason.2030.consequence';
        Meta.Priority := E_Severity.LOW;
        Meta.Category := E_Category.SYSTEM;
        Meta.Shelvable := FALSE;
    33:
        Meta.ReasonCode := 2040;
        Meta.OperatorAction := 'std.reason.2040.action';
        Meta.Consequence := 'std.reason.2040.consequence';
        Meta.Priority := E_Severity.MED;
        Meta.Category := E_Category.SYSTEM;
        Meta.Shelvable := FALSE;
    34:
        Meta.ReasonCode := 2041;
        Meta.OperatorAction := 'std.reason.2041.action';
        Meta.Consequence := 'std.reason.2041.consequence';
        Meta.Priority := E_Severity.MED;
        Meta.Category := E_Category.SYSTEM;
        Meta.Shelvable := FALSE;
    35:
        Meta.ReasonCode := 2042;
        Meta.OperatorAction := 'std.reason.2042.action';
        Meta.Consequence := 'std.reason.2042.consequence';
        Meta.Priority := E_Severity.LOW;
        Meta.Category := E_Category.SYSTEM;
        Meta.Shelvable := FALSE;
    36:
        Meta.ReasonCode := 2043;
        Meta.OperatorAction := '';
        Meta.Consequence := 'std.reason.2043.consequence';
        Meta.Priority := E_Severity.LOW;
        Meta.Category := E_Category.SYSTEM;
        Meta.Shelvable := FALSE;
    37:
        Meta.ReasonCode := 2901;
        Meta.OperatorAction := '';
        Meta.Consequence := 'std.reason.2901.consequence';
        Meta.Priority := E_Severity.LOW;
        Meta.Category := E_Category.SYSTEM;
        Meta.Shelvable := FALSE;
    38:
        Meta.ReasonCode := 10001;
        Meta.OperatorAction := 'std.reason.10001.action';
        Meta.Consequence := 'std.reason.10001.consequence';
        Meta.Priority := E_Severity.MED;
        Meta.Category := E_Category.PROCESS;
        Meta.Shelvable := FALSE;
    39:
        Meta.ReasonCode := 10002;
        Meta.OperatorAction := 'std.reason.10002.action';
        Meta.Consequence := 'std.reason.10002.consequence';
        Meta.Priority := E_Severity.MED;
        Meta.Category := E_Category.PROCESS;
        Meta.Shelvable := FALSE;
    40:
        Meta.ReasonCode := 10003;
        Meta.OperatorAction := 'std.reason.10003.action';
        Meta.Consequence := 'std.reason.10003.consequence';
        Meta.Priority := E_Severity.MED;
        Meta.Category := E_Category.PROCESS;
        Meta.Shelvable := FALSE;
    41:
        Meta.ReasonCode := 10004;
        Meta.OperatorAction := 'std.reason.10004.action';
        Meta.Consequence := 'std.reason.10004.consequence';
        Meta.Priority := E_Severity.MED;
        Meta.Category := E_Category.PROCESS;
        Meta.Shelvable := FALSE;
    42:
        Meta.ReasonCode := 10005;
        Meta.OperatorAction := 'std.reason.10005.action';
        Meta.Consequence := 'std.reason.10005.consequence';
        Meta.Priority := E_Severity.MED;
        Meta.Category := E_Category.PROCESS;
        Meta.Shelvable := FALSE;
    43:
        Meta.ReasonCode := 10101;
        Meta.OperatorAction := 'std.reason.10101.action';
        Meta.Consequence := 'std.reason.10101.consequence';
        Meta.Priority := E_Severity.MED;
        Meta.Category := E_Category.PROCESS;
        Meta.Shelvable := FALSE;
    44:
        Meta.ReasonCode := 10102;
        Meta.OperatorAction := 'std.reason.10102.action';
        Meta.Consequence := 'std.reason.10102.consequence';
        Meta.Priority := E_Severity.MED;
        Meta.Category := E_Category.PROCESS;
        Meta.Shelvable := FALSE;
    45:
        Meta.ReasonCode := 10103;
        Meta.OperatorAction := 'std.reason.10103.action';
        Meta.Consequence := 'std.reason.10103.consequence';
        Meta.Priority := E_Severity.HIGH;
        Meta.Category := E_Category.PROCESS;
        Meta.Shelvable := FALSE;
    46:
        Meta.ReasonCode := 10111;
        Meta.OperatorAction := 'std.reason.10111.action';
        Meta.Consequence := 'std.reason.10111.consequence';
        Meta.Priority := E_Severity.MED;
        Meta.Category := E_Category.PROCESS;
        Meta.Shelvable := FALSE;
    47:
        Meta.ReasonCode := 10112;
        Meta.OperatorAction := 'std.reason.10112.action';
        Meta.Consequence := 'std.reason.10112.consequence';
        Meta.Priority := E_Severity.MED;
        Meta.Category := E_Category.PROCESS;
        Meta.Shelvable := FALSE;
    48:
        Meta.ReasonCode := 10113;
        Meta.OperatorAction := 'std.reason.10113.action';
        Meta.Consequence := 'std.reason.10113.consequence';
        Meta.Priority := E_Severity.HIGH;
        Meta.Category := E_Category.PROCESS;
        Meta.Shelvable := FALSE;
    49:
        Meta.ReasonCode := 10114;
        Meta.OperatorAction := 'std.reason.10114.action';
        Meta.Consequence := 'std.reason.10114.consequence';
        Meta.Priority := E_Severity.MED;
        Meta.Category := E_Category.PROCESS;
        Meta.Shelvable := FALSE;
    50:
        Meta.ReasonCode := 10115;
        Meta.OperatorAction := 'std.reason.10115.action';
        Meta.Consequence := 'std.reason.10115.consequence';
        Meta.Priority := E_Severity.MED;
        Meta.Category := E_Category.SYSTEM;
        Meta.Shelvable := FALSE;
    51:
        Meta.ReasonCode := 10116;
        Meta.OperatorAction := 'std.reason.10116.action';
        Meta.Consequence := 'std.reason.10116.consequence';
        Meta.Priority := E_Severity.MED;
        Meta.Category := E_Category.PROCESS;
        Meta.Shelvable := FALSE;
    52:
        Meta.ReasonCode := 10201;
        Meta.OperatorAction := 'std.reason.10201.action';
        Meta.Consequence := 'std.reason.10201.consequence';
        Meta.Priority := E_Severity.MED;
        Meta.Category := E_Category.PROCESS;
        Meta.Shelvable := FALSE;
    53:
        Meta.ReasonCode := 10202;
        Meta.OperatorAction := 'std.reason.10202.action';
        Meta.Consequence := 'std.reason.10202.consequence';
        Meta.Priority := E_Severity.MED;
        Meta.Category := E_Category.PROCESS;
        Meta.Shelvable := FALSE;
    54:
        Meta.ReasonCode := 10203;
        Meta.OperatorAction := 'std.reason.10203.action';
        Meta.Consequence := 'std.reason.10203.consequence';
        Meta.Priority := E_Severity.HIGH;
        Meta.Category := E_Category.SYSTEM;
        Meta.Shelvable := FALSE;
    55:
        Meta.ReasonCode := 10204;
        Meta.OperatorAction := 'std.reason.10204.action';
        Meta.Consequence := 'std.reason.10204.consequence';
        Meta.Priority := E_Severity.MED;
        Meta.Category := E_Category.PROCESS;
        Meta.Shelvable := FALSE;
    56:
        Meta.ReasonCode := 10205;
        Meta.OperatorAction := 'std.reason.10205.action';
        Meta.Consequence := 'std.reason.10205.consequence';
        Meta.Priority := E_Severity.MED;
        Meta.Category := E_Category.PROCESS;
        Meta.Shelvable := FALSE;
    57:
        Meta.ReasonCode := 10206;
        Meta.OperatorAction := 'std.reason.10206.action';
        Meta.Consequence := 'std.reason.10206.consequence';
        Meta.Priority := E_Severity.LOW;
        Meta.Category := E_Category.PROCESS;
        Meta.Shelvable := FALSE;
    58:
        Meta.ReasonCode := 10301;
        Meta.OperatorAction := 'std.reason.10301.action';
        Meta.Consequence := 'std.reason.10301.consequence';
        Meta.Priority := E_Severity.MED;
        Meta.Category := E_Category.PROCESS;
        Meta.Shelvable := FALSE;
    59:
        Meta.ReasonCode := 10303;
        Meta.OperatorAction := 'std.reason.10303.action';
        Meta.Consequence := 'std.reason.10303.consequence';
        Meta.Priority := E_Severity.HIGH;
        Meta.Category := E_Category.PROCESS;
        Meta.Shelvable := FALSE;
    60:
        Meta.ReasonCode := 10304;
        Meta.OperatorAction := 'std.reason.10304.action';
        Meta.Consequence := 'std.reason.10304.consequence';
        Meta.Priority := E_Severity.HIGH;
        Meta.Category := E_Category.PROCESS;
        Meta.Shelvable := FALSE;
    61:
        Meta.ReasonCode := 10305;
        Meta.OperatorAction := 'std.reason.10305.action';
        Meta.Consequence := 'std.reason.10305.consequence';
        Meta.Priority := E_Severity.MED;
        Meta.Category := E_Category.PROCESS;
        Meta.Shelvable := FALSE;
    62:
        Meta.ReasonCode := 10308;
        Meta.OperatorAction := 'std.reason.10308.action';
        Meta.Consequence := 'std.reason.10308.consequence';
        Meta.Priority := E_Severity.MED;
        Meta.Category := E_Category.PROCESS;
        Meta.Shelvable := FALSE;
    63:
        Meta.ReasonCode := 10310;
        Meta.OperatorAction := 'std.reason.10310.action';
        Meta.Consequence := 'std.reason.10310.consequence';
        Meta.Priority := E_Severity.MED;
        Meta.Category := E_Category.PROCESS;
        Meta.Shelvable := FALSE;
    64:
        Meta.ReasonCode := 10311;
        Meta.OperatorAction := 'std.reason.10311.action';
        Meta.Consequence := 'std.reason.10311.consequence';
        Meta.Priority := E_Severity.MED;
        Meta.Category := E_Category.PROCESS;
        Meta.Shelvable := FALSE;
    65:
        Meta.ReasonCode := 10313;
        Meta.OperatorAction := 'std.reason.10313.action';
        Meta.Consequence := 'std.reason.10313.consequence';
        Meta.Priority := E_Severity.HIGH;
        Meta.Category := E_Category.PROCESS;
        Meta.Shelvable := FALSE;
    66:
        Meta.ReasonCode := 10314;
        Meta.OperatorAction := 'std.reason.10314.action';
        Meta.Consequence := 'std.reason.10314.consequence';
        Meta.Priority := E_Severity.MED;
        Meta.Category := E_Category.PROCESS;
        Meta.Shelvable := FALSE;
    67:
        Meta.ReasonCode := 10315;
        Meta.OperatorAction := 'std.reason.10315.action';
        Meta.Consequence := 'std.reason.10315.consequence';
        Meta.Priority := E_Severity.HIGH;
        Meta.Category := E_Category.PROCESS;
        Meta.Shelvable := FALSE;
    68:
        Meta.ReasonCode := 10401;
        Meta.OperatorAction := 'std.reason.10401.action';
        Meta.Consequence := 'std.reason.10401.consequence';
        Meta.Priority := E_Severity.MED;
        Meta.Category := E_Category.SYSTEM;
        Meta.Shelvable := FALSE;
    69:
        Meta.ReasonCode := 10402;
        Meta.OperatorAction := 'std.reason.10402.action';
        Meta.Consequence := 'std.reason.10402.consequence';
        Meta.Priority := E_Severity.LOW;
        Meta.Category := E_Category.SYSTEM;
        Meta.Shelvable := TRUE;
    70:
        Meta.ReasonCode := 10403;
        Meta.OperatorAction := 'std.reason.10403.action';
        Meta.Consequence := 'std.reason.10403.consequence';
        Meta.Priority := E_Severity.MED;
        Meta.Category := E_Category.SYSTEM;
        Meta.Shelvable := FALSE;
    71:
        Meta.ReasonCode := 10404;
        Meta.OperatorAction := 'std.reason.10404.action';
        Meta.Consequence := 'std.reason.10404.consequence';
        Meta.Priority := E_Severity.LOW;
        Meta.Category := E_Category.SYSTEM;
        Meta.Shelvable := TRUE;
    72:
        Meta.ReasonCode := 10405;
        Meta.OperatorAction := 'std.reason.10405.action';
        Meta.Consequence := 'std.reason.10405.consequence';
        Meta.Priority := E_Severity.MED;
        Meta.Category := E_Category.SYSTEM;
        Meta.Shelvable := FALSE;
    73:
        Meta.ReasonCode := 10406;
        Meta.OperatorAction := 'std.reason.10406.action';
        Meta.Consequence := 'std.reason.10406.consequence';
        Meta.Priority := E_Severity.MED;
        Meta.Category := E_Category.SYSTEM;
        Meta.Shelvable := FALSE;
    74:
        Meta.ReasonCode := 10501;
        Meta.OperatorAction := 'std.reason.10501.action';
        Meta.Consequence := 'std.reason.10501.consequence';
        Meta.Priority := E_Severity.LOW;
        Meta.Category := E_Category.PROCESS;
        Meta.Shelvable := FALSE;
    75:
        Meta.ReasonCode := 10502;
        Meta.OperatorAction := 'std.reason.10502.action';
        Meta.Consequence := 'std.reason.10502.consequence';
        Meta.Priority := E_Severity.HIGH;
        Meta.Category := E_Category.PROCESS;
        Meta.Shelvable := FALSE;
    76:
        Meta.ReasonCode := 10601;
        Meta.OperatorAction := 'std.reason.10601.action';
        Meta.Consequence := 'std.reason.10601.consequence';
        Meta.Priority := E_Severity.MED;
        Meta.Category := E_Category.PROCESS;
        Meta.Shelvable := FALSE;
    77:
        Meta.ReasonCode := 11001;
        Meta.OperatorAction := 'std.reason.11001.action';
        Meta.Consequence := 'std.reason.11001.consequence';
        Meta.Priority := E_Severity.MED;
        Meta.Category := E_Category.PROCESS;
        Meta.Shelvable := FALSE;
ELSE
    RETURN;
END_CASE
F_ReasonMetaByIndex := TRUE;

END_FUNCTION

// ---- Platform/F_TimeSynchronized.TcPOU
// Core §2.7 — quality bit stored with every generated wall-clock record.
FUNCTION F_TimeSynchronized : BOOL

F_TimeSynchronized := GVL_FraktalTime.Current.Available
    AND GVL_FraktalTime.Current.Synchronized;

END_FUNCTION

// ---- BaseClasses/FB_ConfigPager.TcPOU
// Core §3.10.2 — windowed writer for the configuration manifest. QUERY_CONFIG
// re-walks the whole export enumeration each request; the pager counts every
// appended entry and stores only the requested page window into the published
// ST_ConfigPage, so no full manifest buffer ever exists in PLC memory and the
// walk order alone defines the paging. Exporters call M_Append*/ignore paging.
//
// §3.8b — it is ALSO the sink for a parameter-set save, and that is the whole
// point of putting it here. A set is "a projection produced by the same
// deterministic walk that builds the §3.10.2 manifest, keyed per value by
// (Scope, WriteKey)". Making the set a second walk would be a second authority
// on what a station's configuration consists of, and the two would drift the
// first time a module registered a value (§1.1 O9). So M_SetupSetSave puts the
// pager in record mode, the ordinary M_AppendConfig walk runs unchanged, and
// every capability it emits is offered to the store. No exporter knows which
// mode it is feeding, and none can be written to feed only one of them.
FUNCTION_BLOCK FB_ConfigPager
VAR
    {attribute 'OPC.UA.DA' := '0'}
    _pTarget : POINTER TO ST_ConfigPage;
    _cursor  : DINT;   // entries appended so far in this walk
    _first   : DINT;   // first cursor index stored in the window (0-based)
    _storedSlot : INT; // 1-based slot written by the last M_Append; 0 if absent
    // §3.8b set-save mode. Exactly one of _pTarget / _setStore is ever live.
    {attribute 'OPC.UA.DA' := '0'}
    _setStore  : I_ConfigStore;
    _setKind   : E_ConfigKind;
    _setCount  : INT;
    _setFailed : BOOL;
    // §3.8d - the root's access manager, set before a manifest walk. 0 (a pager
    // nobody configured, such as a test's) publishes every value as readable.
    {attribute 'OPC.UA.DA' := '0'}
    _pAccess : POINTER TO FB_AccessManager;
    // §3.8a - another model's page: only model-scoped capabilities are counted
    // and stored. Reset by every M_Setup.
    _modelOnly : BOOL;
END_VAR

; // stateless between requests — driven entirely by M_Setup/M_Append/M_Finish

// §3.8d - the access manager whose policy and session decide what the next
// manifest walk may show. Set by the root before each QUERY_CONFIG.
METHOD M_SetAccess : BOOL
VAR_INPUT
    pAccess : POINTER TO FB_AccessManager;
END_VAR
_pAccess := pAccess;
M_SetAccess := (pAccess <> 0);
END_METHOD

// Begin one QUERY_CONFIG walk targeting the published page window.
METHOD M_Setup : BOOL
VAR_INPUT
    Target    : POINTER TO ST_ConfigPage;
    PageIndex : INT;
    Revision  : UDINT;
END_VAR
M_Setup := FALSE;
_pTarget := 0;
_storedSlot := 0;
_setStore := 0;                 // a manifest walk never writes set records
_modelOnly := FALSE;
IF Target = 0 THEN
    RETURN;
END_IF
_pTarget := Target;
_cursor := 0;
IF PageIndex < 0 THEN
    _first := 0;
ELSE
    _first := TO_DINT(PageIndex) * TO_DINT(PL_Fraktal.MAX_CONFIG_PAGE);
END_IF
_pTarget^.Revision := Revision;
_pTarget^.PageIndex := SEL(PageIndex < 0, PageIndex, 0);
_pTarget^.PageCount := 0;
_pTarget^.EntryCount := 0;
M_Setup := TRUE;
END_METHOD

// Append one manifest entry; stored only when it falls inside the page window.
// Always returns TRUE so exporters can chain without branching.
METHOD M_Append : BOOL
VAR_INPUT
    Scope     : STRING(255);
    Item      : STRING(255);
    ValueText : STRING(255);
END_VAR
M_Append := TRUE;
_storedSlot := 0;
// Another model's page holds its model data only; a plain entry is none.
IF _modelOnly THEN
    RETURN;
END_IF
_M_Window(Scope := Scope, Item := Item, ValueText := ValueText);
END_METHOD

// Count one entry of the walk and store it when it falls in the page window.
METHOD PRIVATE _M_Window
VAR_INPUT
    Scope     : STRING(255);
    Item      : STRING(255);
    ValueText : STRING(255);
END_VAR
VAR
    slot : DINT;
END_VAR
_storedSlot := 0;
IF _pTarget = 0 THEN
    RETURN;
END_IF
slot := _cursor - _first;   // window-relative 0-based position
_cursor := _cursor + 1;
IF (slot < 0) OR (slot >= TO_DINT(PL_Fraktal.MAX_CONFIG_PAGE)) THEN
    RETURN;                 // outside the requested window — counted, not stored
END_IF
_pTarget^.Entries[TO_INT(slot) + 1].Scope := Scope;
_pTarget^.Entries[TO_INT(slot) + 1].Item := Item;
_pTarget^.Entries[TO_INT(slot) + 1].ValueText := ValueText;
// Explicitly clear the capability tail so a reused response slot cannot retain
// write authority from an earlier page.
_pTarget^.Entries[TO_INT(slot) + 1].WriteKey := '';
_pTarget^.Entries[TO_INT(slot) + 1].WriteRevision := 0;
_pTarget^.Entries[TO_INT(slot) + 1].ConfigKind := E_ConfigKind.PAR_CFG;
_pTarget^.Entries[TO_INT(slot) + 1].ValueType := E_ConfigValueType.TEXT;
_pTarget^.Entries[TO_INT(slot) + 1].Writable := FALSE;
_pTarget^.Entries[TO_INT(slot) + 1].RequiresReady := FALSE;
_pTarget^.Entries[TO_INT(slot) + 1].HasMinimum := FALSE;
_pTarget^.Entries[TO_INT(slot) + 1].HasMaximum := FALSE;
_pTarget^.Entries[TO_INT(slot) + 1].Minimum := 0.0;
_pTarget^.Entries[TO_INT(slot) + 1].Maximum := 0.0;
_pTarget^.Entries[TO_INT(slot) + 1].Unit := '';
_pTarget^.Entries[TO_INT(slot) + 1].LabelKey := '';
_pTarget^.Entries[TO_INT(slot) + 1].EnumDomain := '';
_pTarget^.Entries[TO_INT(slot) + 1].UnitCode := E_EngUnit.NONE;
_pTarget^.Entries[TO_INT(slot) + 1].EnumLabelKey := '';
_pTarget^.Entries[TO_INT(slot) + 1].ClassId := '';
_pTarget^.Entries[TO_INT(slot) + 1].ReadLevel := E_AccessLevel.NONE;
_pTarget^.Entries[TO_INT(slot) + 1].WriteLevel := E_AccessLevel.NONE;
_pTarget^.Entries[TO_INT(slot) + 1].Readable := TRUE;
_pTarget^.Entries[TO_INT(slot) + 1].ModelScoped := FALSE;
// §3.8d - a plain (non-capability) entry is readable at DATA_READ.
IF _pAccess <> 0 THEN
    _pTarget^.Entries[TO_INT(slot) + 1].ReadLevel :=
        _pAccess^.M_DataLevel(ClassId := '', MinLevel := E_AccessLevel.NONE, ForWrite := FALSE);
    IF NOT _pAccess^.M_PermitsLevel(Required := _pTarget^.Entries[TO_INT(slot) + 1].ReadLevel) THEN
        _pTarget^.Entries[TO_INT(slot) + 1].ValueText := '';
        _pTarget^.Entries[TO_INT(slot) + 1].Readable := FALSE;
    END_IF
END_IF
_storedSlot := TO_INT(slot) + 1;
_pTarget^.EntryCount := TO_INT(slot) + 1;
END_METHOD

// Append one typed configuration-write capability. All inputs are explicit for
// TwinCAT 4024 compatibility. The owning handler remains authoritative.
METHOD M_AppendCapability : BOOL
VAR_INPUT
    Scope         : STRING(255);
    Item          : STRING(255);
    ValueText     : STRING(255);
    WriteKey      : STRING(160);
    WriteRevision : UDINT;
    ConfigKind    : E_ConfigKind;
    ValueType     : E_ConfigValueType;
    Writable      : BOOL;
    RequiresReady : BOOL;
    HasMinimum    : BOOL;
    HasMaximum    : BOOL;
    Minimum       : LREAL;
    Maximum       : LREAL;
    Unit          : E_EngUnit;
    LabelKey      : STRING(160);
    EnumDomain    : STRING(255);
    EnumLabelKey  : STRING(80);
    ClassId       : STRING(40);    // §3.8d; '' = built-in class
    MinReadLevel  : E_AccessLevel;
    MinWriteLevel : E_AccessLevel;
    ModelScoped   : BOOL;          // Core 0.19 - follows the model a request names
END_VAR
VAR
    readLevel  : E_AccessLevel;
    writeLevel : E_AccessLevel;
    readable   : BOOL;
END_VAR
M_AppendCapability := TRUE;
_storedSlot := 0;
IF _modelOnly THEN
    IF NOT ModelScoped THEN
        RETURN;
    END_IF
    _M_Window(Scope := Scope, Item := Item, ValueText := ValueText);
ELSE
    M_AppendCapability := M_Append(Scope := Scope, Item := Item,
        ValueText := ValueText);
END_IF
// §3.8b — offered to an open set save BEFORE the page-window test, because a
// set has no window: it takes every record the walk produces, whichever page
// the same walk would have put it on.
_M_OfferRecord(Scope := Scope, ValueText := ValueText, WriteKey := WriteKey,
    WriteRevision := WriteRevision, ConfigKind := ConfigKind,
    ValueType := ValueType, Writable := Writable);
IF (_pTarget = 0) OR (_storedSlot <= 0) THEN
    RETURN;
END_IF
_pTarget^.Entries[_storedSlot].WriteKey := WriteKey;
_pTarget^.Entries[_storedSlot].WriteRevision := WriteRevision;
_pTarget^.Entries[_storedSlot].ConfigKind := ConfigKind;
_pTarget^.Entries[_storedSlot].ValueType := ValueType;
_pTarget^.Entries[_storedSlot].Writable := Writable
    AND (WriteKey <> '') AND (WriteRevision > 0);
_pTarget^.Entries[_storedSlot].RequiresReady := RequiresReady;
_pTarget^.Entries[_storedSlot].HasMinimum := HasMinimum;
_pTarget^.Entries[_storedSlot].HasMaximum := HasMaximum;
_pTarget^.Entries[_storedSlot].Minimum := Minimum;
_pTarget^.Entries[_storedSlot].Maximum := Maximum;
_pTarget^.Entries[_storedSlot].Unit := F_EngUnitSymbol(Unit := Unit);
_pTarget^.Entries[_storedSlot].UnitCode := Unit;
_pTarget^.Entries[_storedSlot].LabelKey := LabelKey;
_pTarget^.Entries[_storedSlot].EnumDomain := EnumDomain;
_pTarget^.Entries[_storedSlot].EnumLabelKey := EnumLabelKey;
_pTarget^.Entries[_storedSlot].ModelScoped := ModelScoped;
// §3.8d - effective levels, computed once and before the value is placed, so a
// class that is readable below DATA_READ shows its value and one that is not
// never does. The set record above was offered the real value regardless: a
// save reveals nothing outside the PLC.
readLevel := MinReadLevel;
writeLevel := MinWriteLevel;
readable := TRUE;
IF _pAccess <> 0 THEN
    readLevel := _pAccess^.M_DataLevel(ClassId := ClassId, MinLevel := MinReadLevel,
        ForWrite := FALSE);
    writeLevel := _pAccess^.M_DataLevel(ClassId := ClassId, MinLevel := MinWriteLevel,
        ForWrite := TRUE);
    readable := _pAccess^.M_PermitsLevel(Required := readLevel);
END_IF
_pTarget^.Entries[_storedSlot].ClassId := ClassId;
_pTarget^.Entries[_storedSlot].ReadLevel := readLevel;
_pTarget^.Entries[_storedSlot].WriteLevel := writeLevel;
_pTarget^.Entries[_storedSlot].Readable := readable;
IF readable THEN
    _pTarget^.Entries[_storedSlot].ValueText := ValueText;
ELSE
    _pTarget^.Entries[_storedSlot].ValueText := '';
END_IF
END_METHOD

// §3.8b — offer one capability to an open set save. Called from
// M_AppendCapability, so the set contains exactly what the manifest publishes
// as editable and nothing else: no unregistered value can enter a set, and no
// registered one can be forgotten by it.
//
// Only records of the set's own ConfigKind are taken — a station set carries
// STATION_CFG, a model set carries PAR_CFG (§3.8b "one mechanism, two kinds").
// Anything that will not fit a record FAILS the save rather than shortening a
// value: a set that quietly lost a character restores a machine to almost its
// commissioned state, which is worse than not restoring it.
METHOD PRIVATE _M_OfferRecord
VAR_INPUT
    Scope         : STRING(255);
    ValueText     : STRING(255);
    WriteKey      : STRING(160);
    WriteRevision : UDINT;
    ConfigKind    : E_ConfigKind;
    ValueType     : E_ConfigValueType;
    Writable      : BOOL;
END_VAR
VAR
    record : ST_ConfigRecord;
END_VAR
IF _setStore = 0 THEN
    RETURN;
END_IF
IF _setFailed THEN
    RETURN;                     // a failed transaction takes no further records
END_IF
IF NOT Writable THEN
    RETURN;                     // read-only publication is not configuration
END_IF
IF (WriteKey = '') OR (WriteRevision = 0) THEN
    RETURN;                     // fails closed exactly as the manifest does
END_IF
IF ConfigKind <> _setKind THEN
    RETURN;                     // the other kind of set owns this record
END_IF
IF TO_INT(LEN(Scope)) > 80 THEN
    _setFailed := TRUE;
    RETURN;
END_IF
IF TO_INT(LEN(ValueText)) > 80 THEN
    _setFailed := TRUE;
    RETURN;
END_IF
record.Scope := Scope;
record.WriteKey := WriteKey;
record.Revision := WriteRevision;
record.Kind := ConfigKind;
record.ValueType := ValueType;
record.ValueText := ValueText;
IF _setStore.M_SaveRecord(Record := record) THEN
    _setCount := _setCount + 1;
ELSE
    _setFailed := TRUE;
END_IF
END_METHOD

// §3.8b — begin a parameter-set save. The caller then runs the ordinary
// M_AppendConfig walk and closes with M_FinishSetSave.
METHOD M_SetupSetSave : BOOL
VAR_INPUT
    Store : I_ConfigStore;
    Info  : ST_ConfigSetInfo;
END_VAR
M_SetupSetSave := FALSE;
_pTarget := 0;                  // a set walk never writes a manifest page
_storedSlot := 0;
_setStore := 0;
_setCount := 0;
_setFailed := FALSE;
_modelOnly := FALSE;
IF Store = 0 THEN
    RETURN;
END_IF
IF NOT Store.M_SaveBegin(Info := Info) THEN
    RETURN;
END_IF
_setStore := Store;
_setKind := Info.Kind;
M_SetupSetSave := TRUE;
END_METHOD

// §3.8b — close the set save. FALSE means nothing was stored: an empty set, a
// record that would not fit, or a store that refused the commit. The previous
// set of that name is left exactly as it was.
METHOD M_FinishSetSave : BOOL
VAR_OUTPUT
    Records : INT;
END_VAR
VAR
    store : I_ConfigStore;
END_VAR
M_FinishSetSave := FALSE;
Records := _setCount;
store := _setStore;
_setStore := 0;
IF store = 0 THEN
    RETURN;
END_IF
IF _setFailed OR (_setCount = 0) THEN
    // An empty set is refused rather than stored: a named set that restores
    // nothing is the one somebody loads believing it did something.
    store.M_SaveAbort();
    RETURN;
END_IF
M_FinishSetSave := store.M_SaveCommit();
END_METHOD

METHOD M_AppendNumber : BOOL
VAR_INPUT
    Scope  : STRING(255);
    Item   : STRING(255);
    Number : DINT;
END_VAR
M_AppendNumber := M_Append(Scope := Scope, Item := Item,
    ValueText := TO_STRING(Number));
// Declare the type the caller already knows. M_Append stores every entry as
// TEXT, so without this the number crosses the wire indistinguishable from a
// string and the consumer has to guess from the leaf NAME. The HMI did exactly
// that, against a hand-maintained allowlist that did not include StepNo — so
// every §3.13 flow-chart row rendered as "N0" with an empty drill-down while
// the value was sitting there as the string "100". A type the sender knows
// must never be re-derived by the receiver.
IF (_pTarget <> 0) AND (_storedSlot > 0) THEN
    _pTarget^.Entries[_storedSlot].ValueType := E_ConfigValueType.NUMBER;
END_IF
END_METHOD

// §3.8a - the rest of this walk serves another model's record: only
// capabilities marked ModelScoped are counted and stored, so the answer is that
// model's data - a page or two - not the whole station manifest.
METHOD M_SetModelOnly : BOOL
VAR_INPUT
    Enabled : BOOL;
END_VAR
_modelOnly := Enabled;
M_SetModelOnly := TRUE;
END_METHOD

// Close the walk: publish the total page count for the HMI's fetch loop.
METHOD M_Finish : BOOL
M_Finish := FALSE;
IF _pTarget = 0 THEN
    RETURN;
END_IF
_pTarget^.PageCount := TO_INT(
    (_cursor + TO_DINT(PL_Fraktal.MAX_CONFIG_PAGE) - 1)
    / TO_DINT(PL_Fraktal.MAX_CONFIG_PAGE));
M_Finish := TRUE;
END_METHOD

END_FUNCTION_BLOCK

// ---- BaseClasses/FB_AccessManager.TcPOU
// Core §7.7(c) — per-root session + enforcement. Login/logout is DATA-DRIVEN
// (§3.10(a')): the HMI writes ReqUser/ReqSecret and pulses ReqLogin/ReqLogout;
// the secret is cleared after every attempt. Policy default: fully open (§7.7(b)).
FUNCTION_BLOCK FB_AccessManager
VAR_INPUT
    ReqUser   : STRING(32);          // HMI-writable login request
    ReqSecret : STRING(32);          // cleared after each attempt (§7.7(c))
    ReqLogin  : BOOL;
    ReqLogout : BOOL;
END_VAR
VAR_OUTPUT
    SessionGeneration : UDINT; // changes on every successful login/session termination
    CurrentUser  : STRING(32);
    CurrentLevel : E_AccessLevel;    // HMI greys controls from this; PLC re-checks
    LoginFailed  : BOOL;             // last attempt outcome (HMI feedback)
END_VAR
VAR PERSISTENT
    Policy : ST_AccessPolicy;
    // §3.8d - data-class levels. A SEPARATE persistent table on purpose: adding
    // members to Policy would change its layout, TwinCAT would reinitialize it on
    // the next download, and a locked-down station would silently come back
    // fully open. A new variable starts empty and touches nothing that exists.
    ClassCount : INT;
    Classes    : ARRAY[1..PL_Fraktal.MAX_DATA_CLASSES] OF ST_DataClassPolicy;        // §3.8a station config; edit gated by ACCESS_POLICY
END_VAR
VAR
    {attribute 'OPC.UA.DA' := '0'}
    _provider : I_AccessProvider;
    {attribute 'OPC.UA.DA' := '0'}
    _log      : POINTER TO FB_AlarmLog;
    _tIdle    : TON;
    _activityPending : BOOL;          // accepted operator action rearms the idle timer
    // §7.7(c) - the provider's durable-table service, when it offers one.
    {attribute 'OPC.UA.DA' := '0'}
    _store : I_AccessStore;
    _storeRestored : BOOL;              // the store's table has been read
    _restoreLossSeen : BOOL;          // this root has taken the provider's loss
    _restoreLossTake : BOOL;          // pending for the root's §3.8b annunciation
    _saveFailedSlot : INT;            // open CONFIG_PERSIST_FAILED event (0 = none)
END_VAR

// event/session handling is in Cyclic (called by the owning Unit each scan)

METHOD Cyclic : BOOL
VAR
    lvl : E_AccessLevel;
    loginHandled : BOOL;
    logoutHandled : BOOL;
    sessionRearm : BOOL;
    activityHandled : BOOL;
END_VAR
// §7.7(c) - restore/save the provider's table before this scan's login, so a
// restored user can log in on the scan the table arrives.
IF _store <> 0 THEN
    _storeRestored := _store.M_Service();
    _M_StoreCyclic();
END_IF
sessionRearm := FALSE;
loginHandled := ReqLogin;
IF loginHandled THEN
    ReqLogin := FALSE;
    lvl := E_AccessLevel.NONE;
    IF _provider <> 0 THEN
        lvl := _provider.Authenticate(User := ReqUser, Secret := ReqSecret);
    END_IF
    ReqSecret := '';                                   // never retain the secret
    IF lvl > E_AccessLevel.NONE THEN
        SessionGeneration := SessionGeneration + 1;
        CurrentUser := ReqUser;
        CurrentLevel := lvl;
        LoginFailed := FALSE;
        sessionRearm := TRUE;
        _M_Audit('std.audit.login', CurrentUser);
    ELSE
        LoginFailed := TRUE;
        _M_Audit('std.audit.loginFailed', ReqUser);
    END_IF
END_IF
logoutHandled := ReqLogout;
IF logoutHandled THEN
    ReqLogout := FALSE;
    SessionGeneration := SessionGeneration + 1;
    IF CurrentLevel > E_AccessLevel.NONE THEN
        _M_Audit('std.audit.logout', CurrentUser);
        CurrentUser := '';
        CurrentLevel := E_AccessLevel.NONE;
    END_IF
END_IF
// Idle means time since the last accepted authenticated operator action, not
// absolute session age. Background reads/release queries never call RecordActivity.
activityHandled := _activityPending;
_activityPending := FALSE;
_tIdle(IN := (Policy.SessionTimeout > T#0S)
       AND (CurrentLevel > E_AccessLevel.NONE)
       AND NOT sessionRearm AND NOT activityHandled,
       PT := Policy.SessionTimeout);
IF _tIdle.Q THEN
    _M_Audit('std.audit.autoLogout', CurrentUser);
    SessionGeneration := SessionGeneration + 1;
        CurrentUser := '';
    CurrentLevel := E_AccessLevel.NONE;
END_IF
Cyclic := TRUE;
END_METHOD

// Startup/station-configuration seam; runtime HMI writes remain Unit-gated.
METHOD ConfigureRequired : BOOL
VAR_INPUT
    Gate : E_GatedAction;
    Level : E_AccessLevel;
END_VAR
// Upper bound = the LAST E_GatedAction member; it moves with every appended gate.
IF (TO_INT(Gate) < 0) OR (TO_INT(Gate) > TO_INT(E_GatedAction.CONFIG_SET))
OR (TO_INT(Level) < TO_INT(E_AccessLevel.NONE)) OR (TO_INT(Level) > TO_INT(E_AccessLevel.ADMIN)) THEN
    ConfigureRequired := FALSE;
ELSE
    Policy.Required[TO_INT(Gate)] := Level;
    ConfigureRequired := TRUE;
END_IF
END_METHOD

// Persistent station-policy edit. Seven days is a defensive upper bound that
// stays within the signed millisecond TIME conversion used by the TC3 binding.
METHOD ConfigureSessionTimeout : BOOL
VAR_INPUT
    TimeoutMs : UDINT;
END_VAR
IF TimeoutMs > 604800000 THEN
    ConfigureSessionTimeout := FALSE;
    RETURN;
END_IF
Policy.SessionTimeout := DINT_TO_TIME(TO_DINT(TimeoutMs));
ConfigureSessionTimeout := TRUE;
END_METHOD

// ST-facing request seam. OPC UA clients continue to write the published request data.
METHOD RequestLogin : BOOL
VAR_INPUT
    User : STRING(32);
    Secret : STRING(32);
END_VAR
ReqUser := User;
ReqSecret := Secret;
ReqLogin := TRUE;
RequestLogin := TRUE;
END_METHOD

// ST-facing request seam; the cyclic edge handler performs the state change and audit.
METHOD RequestLogout : BOOL
ReqLogout := TRUE;
RequestLogout := TRUE;
END_METHOD

// Called only by accepted gated operator actions. Keeping this explicit prevents
// periodic reads and release-panel polling from keeping an abandoned session alive.
METHOD RecordActivity : BOOL
RecordActivity := CurrentLevel > E_AccessLevel.NONE;
IF RecordActivity THEN
    _activityPending := TRUE;
END_IF
END_METHOD

// pure check for UI/logic — no logging
METHOD Permits : BOOL
VAR_INPUT
    Gate : E_GatedAction;
END_VAR
Permits := FALSE;
// Upper bound = the LAST E_GatedAction member. It said POWER_CONTROL after
// CONFIG_SET was appended, so every parameter-set operation was refused.
IF (TO_INT(Gate) < 0) OR (TO_INT(Gate) > TO_INT(E_GatedAction.CONFIG_SET)) THEN
    RETURN;
END_IF
IF (TO_INT(CurrentLevel) < TO_INT(E_AccessLevel.NONE)) OR (TO_INT(CurrentLevel) > TO_INT(E_AccessLevel.ADMIN)) THEN
    RETURN;
END_IF
IF (TO_INT(Policy.Required[TO_INT(Gate)]) < TO_INT(E_AccessLevel.NONE))
OR (TO_INT(Policy.Required[TO_INT(Gate)]) > TO_INT(E_AccessLevel.ADMIN)) THEN
    RETURN;                                      // corrupt policy fails closed
END_IF
Permits := TO_DINT(CurrentLevel) >= TO_DINT(Policy.Required[TO_INT(Gate)]);
END_METHOD

// §3.8d - the EFFECTIVE level to read or write a value: its class's level,
// raised (never lowered) by the value's own minimum. '' is the built-in class,
// whose levels are the DATA_READ/DATA_WRITE thresholds. An undeclared class or
// a corrupt level fails closed at ADMIN.
METHOD M_DataLevel : E_AccessLevel
VAR_INPUT
    ClassId  : STRING(40);
    MinLevel : E_AccessLevel;
    ForWrite : BOOL;
END_VAR
VAR
    i     : INT;
    n     : INT;
    level : E_AccessLevel;
END_VAR
level := E_AccessLevel.ADMIN;
IF ClassId = '' THEN
    IF ForWrite THEN
        level := Policy.Required[TO_INT(E_GatedAction.DATA_WRITE)];
    ELSE
        level := Policy.Required[TO_INT(E_GatedAction.DATA_READ)];
    END_IF
ELSE
    n := LIMIT(0, ClassCount, PL_Fraktal.MAX_DATA_CLASSES);
    FOR i := 1 TO n DO
        IF Classes[i].ClassId = ClassId THEN
            IF ForWrite THEN
                level := Classes[i].WriteLevel;
            ELSE
                level := Classes[i].ReadLevel;
            END_IF
            EXIT;
        END_IF
    END_FOR
END_IF
IF (TO_DINT(level) < TO_DINT(E_AccessLevel.NONE))
OR (TO_DINT(level) > TO_DINT(E_AccessLevel.ADMIN)) THEN
    level := E_AccessLevel.ADMIN;                // corrupt policy fails closed
END_IF
IF (TO_DINT(MinLevel) < TO_DINT(E_AccessLevel.NONE))
OR (TO_DINT(MinLevel) > TO_DINT(E_AccessLevel.ADMIN)) THEN
    level := E_AccessLevel.ADMIN;
ELSIF TO_DINT(MinLevel) > TO_DINT(level) THEN
    level := MinLevel;                           // raise-only
END_IF
M_DataLevel := level;
END_METHOD

// Pure check of the session against an already-resolved level.
METHOD M_PermitsLevel : BOOL
VAR_INPUT
    Required : E_AccessLevel;
END_VAR
M_PermitsLevel := (TO_DINT(Required) >= TO_DINT(E_AccessLevel.NONE))
    AND (TO_DINT(Required) <= TO_DINT(E_AccessLevel.ADMIN))
    AND (TO_DINT(CurrentLevel) >= TO_DINT(Required));
END_METHOD

// Gated-entry form of M_PermitsLevel: a refusal is audited like a refused
// gated action (§7.7(c)), so a value refused by its class leaves the same trace.
METHOD M_PermitsLevelLogged : BOOL
VAR_INPUT
    Required : E_AccessLevel;
END_VAR
M_PermitsLevelLogged := M_PermitsLevel(Required := Required);
IF NOT M_PermitsLevelLogged THEN
    _M_Audit(What := 'std.audit.dataAccessDenied', Who := CurrentUser);
END_IF
END_METHOD

// §3.8d - declare a data class, normally at Setup on every boot. The levels
// are DEFAULTS: a class already in the persistent table keeps the levels a
// deployment edited, and only its label follows the code. Refused when the
// table is full, the id is empty, or a level is out of range.
METHOD M_DeclareClass : BOOL
VAR_INPUT
    ClassId    : STRING(80);
    LabelKey   : STRING(160);
    ReadLevel  : E_AccessLevel;
    WriteLevel : E_AccessLevel;
END_VAR
VAR
    i : INT;
    n : INT;
END_VAR
M_DeclareClass := FALSE;
IF (ClassId = '') OR (LEN(ClassId) > 40)
OR (TO_DINT(ReadLevel) < TO_DINT(E_AccessLevel.NONE))
OR (TO_DINT(ReadLevel) > TO_DINT(E_AccessLevel.ADMIN))
OR (TO_DINT(WriteLevel) < TO_DINT(E_AccessLevel.NONE))
OR (TO_DINT(WriteLevel) > TO_DINT(E_AccessLevel.ADMIN)) THEN
    RETURN;
END_IF
n := LIMIT(0, ClassCount, PL_Fraktal.MAX_DATA_CLASSES);
ClassCount := n;
FOR i := 1 TO n DO
    IF Classes[i].ClassId = ClassId THEN
        Classes[i].LabelKey := LabelKey;          // the persisted levels stand
        M_DeclareClass := TRUE;
        RETURN;
    END_IF
END_FOR
IF n >= PL_Fraktal.MAX_DATA_CLASSES THEN
    RETURN;
END_IF
n := n + 1;
Classes[n].ClassId := ClassId;
Classes[n].LabelKey := LabelKey;
Classes[n].ReadLevel := ReadLevel;
Classes[n].WriteLevel := WriteLevel;
ClassCount := n;
M_DeclareClass := TRUE;
END_METHOD

// §3.8d/§7.7(b) - change a declared class's read or write level. The caller
// (the root) owns the ACCESS_POLICY gate; this validates and stores only.
METHOD M_SetClassLevel : BOOL
VAR_INPUT
    ClassId  : STRING(80);
    Level    : E_AccessLevel;
    ForWrite : BOOL;
END_VAR
VAR
    i : INT;
    n : INT;
END_VAR
M_SetClassLevel := FALSE;
IF (TO_DINT(Level) < TO_DINT(E_AccessLevel.NONE))
OR (TO_DINT(Level) > TO_DINT(E_AccessLevel.ADMIN)) THEN
    RETURN;
END_IF
n := LIMIT(0, ClassCount, PL_Fraktal.MAX_DATA_CLASSES);
FOR i := 1 TO n DO
    IF Classes[i].ClassId = ClassId THEN
        IF ForWrite THEN
            Classes[i].WriteLevel := Level;
        ELSE
            Classes[i].ReadLevel := Level;
        END_IF
        M_SetClassLevel := TRUE;
        RETURN;
    END_IF
END_FOR
END_METHOD

// gated-entry check: a DENIED attempt is audited as a MESSAGE event (§8.3/§7.7(c))
METHOD PermitsLogged : BOOL
VAR_INPUT
    Gate : E_GatedAction;
END_VAR
PermitsLogged := Permits(Gate := Gate);
IF NOT PermitsLogged THEN
    _M_AuditDenied(Gate := Gate);
END_IF
END_METHOD

METHOD Setup : BOOL
VAR_INPUT
    Provider : I_AccessProvider;
    pAlarmLog : POINTER TO FB_AlarmLog;
END_VAR
IF Provider <> 0 THEN
    _provider := Provider;                  // Unit OnInit may attach only the audit log
    _store := 0;
    __QUERYINTERFACE(Provider, _store);     // optional: a provider that retains its table
END_IF
_log := pAlarmLog;
Setup := TRUE;
END_METHOD

// §3.8b/§7.7(c) - TRUE exactly once per loss: the provider's retained user table
// was rejected or missing at restore. The owning root announces it like any
// other lost configuration image; taking it here never clears the provider.
METHOD M_TakeRestoreLoss : BOOL
M_TakeRestoreLoss := _restoreLossTake;
_restoreLossTake := FALSE;
END_METHOD

// A registration that cannot be written is live now and lost at the next
// restart, so it stands as CONFIG_PERSIST_FAILED until a later write succeeds; a
// retained table that cannot be read stands the same way until it can.
METHOD PRIVATE _M_StoreCyclic
VAR
    text : STRING(80);
END_VAR
IF _store.M_RestoreLost() THEN
    IF NOT _restoreLossSeen THEN
        _restoreLossSeen := TRUE;
        _restoreLossTake := TRUE;
    END_IF
END_IF
IF _store.M_SaveFailed() THEN
    IF (_saveFailedSlot = 0) AND (_log <> 0) THEN
        text := 'std.error.accessPersistFailed';
        IF NOT _storeRestored THEN
            text := 'std.error.storageUnreadable';
        END_IF
        _saveFailedSlot := _log^.Raise(Reason := E_Reason.CONFIG_PERSIST_FAILED,
            Text := text, Source := 'Access',
            Severity := E_Severity.MED, Category := E_Category.SYSTEM,
            ResetClass := E_ResetClass.AUTO_RESET);
    END_IF
ELSIF _saveFailedSlot > 0 THEN
    IF _log <> 0 THEN
        _log^.Gone(Slot := _saveFailedSlot);
    END_IF
    _saveFailedSlot := 0;
END_IF
END_METHOD

// audit trail for free: come+gone MESSAGE lands in the §8.3 ring
METHOD PRIVATE _M_Audit
VAR_INPUT
    What : STRING(64);
    Who : STRING(32);
END_VAR
VAR
    auditSlot : INT;
    txt : STRING(255);
END_VAR
IF _log = 0 THEN
    RETURN;
END_IF
txt := CONCAT(What, ': ');
txt := CONCAT(txt, Who);
auditSlot := _log^.Raise(Reason := E_Reason.NONE, Text := txt,
                 Source := 'Access', Severity := E_Severity.LOW,
                 Category := E_Category.SYSTEM, ResetClass := E_ResetClass.AUTO_RESET);
IF auditSlot > 0 THEN
    _log^.Gone(Slot := auditSlot);                     // instant come+gone -> ring entry
END_IF
END_METHOD

// Include the action ordinal: a generic "denied" record is not actionable audit.
METHOD PRIVATE _M_AuditDenied
VAR_INPUT
    Gate : E_GatedAction;
END_VAR
VAR
    detail : STRING(32);
END_VAR
detail := CONCAT(CurrentUser, ' gate=');
detail := CONCAT(detail, TO_STRING(TO_DINT(Gate)));
_M_Audit(What := 'std.audit.accessDenied', Who := detail);
END_METHOD

END_FUNCTION_BLOCK

// ---- BaseClasses/FB_AlarmLog.TcPOU
// Core §8.3 — per-Unit alarm & event log: active list + closed ring, durations,
// AUTO/MANUAL reset classes, optional historian sink. Fixed-size, never allocates.
FUNCTION_BLOCK FB_AlarmLog
VAR_OUTPUT
    Active    : ARRAY[1..PL_Fraktal.MAX_ALARM_ACTIVE] OF ST_AlarmEvent;  // ACTIVE/WAIT_RESET
    NActive   : INT;
    Ring      : ARRAY[1..PL_Fraktal.MAX_ALARM_RING] OF ST_AlarmEvent;    // closed, newest at RingHead
    RingHead  : INT;
    Blocking  : BOOL;    // any MANUAL_RESET event ACTIVE/WAIT_RESET (§8.3(b))
    Truncated : BOOL;
    // §3.10.2 — rationalization records are static config; excluded from the
    // cyclic OPC UA tree (served via the manifest when an HMI needs them).
    {attribute 'OPC.UA.DA' := '0'}
    Meta      : ARRAY[1..PL_Fraktal.MAX_ALARM_META] OF ST_AlarmMeta;  // §8.9 rationalization
    {attribute 'OPC.UA.DA' := '0'}
    MetaCount : INT;
END_VAR
VAR
    {attribute 'OPC.UA.DA' := '0'}
    _sink    : I_EventSink;
    _comeMs  : ARRAY[1..PL_Fraktal.MAX_ALARM_ACTIVE] OF DWORD;   // monotonic (TC3 §8.11)
    _shelfMs : ARRAY[1..PL_Fraktal.MAX_ALARM_ACTIVE] OF UDINT;   // §8.10 countdown (0 = not shelved)
    _cycLast : TIME;                                             // Cyclic delta stamp
END_VAR

// event-driven; no cyclic body

// §8.3(c) — open a non-channel-specific event; returns slot (0 = full).
METHOD Raise : INT
VAR_INPUT
    Reason : E_Reason;
    Text : STRING(255);
    Source : STRING(255);
    Severity : E_Severity;
    Category : E_Category;
    ResetClass : E_ResetClass;
END_VAR
Raise := _M_Raise(Reason := Reason, Text := Text, Source := Source,
    IoTag := '', IoAddress := '', Severity := Severity, Category := Category,
    ResetClass := ResetClass);
END_METHOD

// §8.3(c) — open an event; returns its slot id (0 = table full -> Truncated)
METHOD PRIVATE _M_Raise : INT
VAR_INPUT
    Reason : E_Reason;
    Text : STRING(255);
    Source : STRING(255);
    IoTag : STRING(80);
    IoAddress : STRING(80);
    Severity : E_Severity;
    Category : E_Category;
    ResetClass : E_ResetClass;
END_VAR
VAR
    i, slot : INT;
    generatedMeta : ST_AlarmMeta;
    effectiveSeverity : E_Severity;
    effectiveCategory : E_Category;
END_VAR
slot := 0;
effectiveSeverity := Severity;
effectiveCategory := Category;
// §8.9: a registered standard reason has one generated priority/class on every
// surface. Unknown project reasons retain the explicit caller values and must
// provide their own runtime rationalization through RegisterMetaFull.
IF F_ReasonMeta(Reason := Reason, Meta := generatedMeta) THEN
    effectiveSeverity := generatedMeta.Priority;
    effectiveCategory := generatedMeta.Category;
ELSE
    FOR i := 1 TO MetaCount DO
        IF Meta[i].ReasonCode = Reason THEN
            effectiveSeverity := Meta[i].Priority;
            effectiveCategory := Meta[i].Category;
            EXIT;
        END_IF
    END_FOR
END_IF
FOR i := 1 TO PL_Fraktal.MAX_ALARM_ACTIVE DO
    IF Active[i].State = E_AlarmState.CLOSED THEN
        slot := i;
        EXIT;
    END_IF
END_FOR
IF slot = 0 THEN
    Truncated := TRUE;
    _M_Raise := 0;
    RETURN;
END_IF
Active[slot].ReasonCode  := Reason;
Active[slot].Description := Text;
Active[slot].SourcePath  := Source;
Active[slot].IoTag       := IoTag;
Active[slot].IoAddress   := IoAddress;
Active[slot].Severity    := effectiveSeverity;
Active[slot].Category    := effectiveCategory;
Active[slot].ResetClass  := ResetClass;
Active[slot].State       := E_AlarmState.ACTIVE;
Active[slot].ComeAt      := F_Now();
Active[slot].ComeTimeSynchronized := F_TimeSynchronized();
Active[slot].GoneAt      := DT#1970-01-01-00:00:00;
Active[slot].ResetAt     := DT#1970-01-01-00:00:00;
Active[slot].GoneTimeSynchronized := FALSE;
Active[slot].ResetTimeSynchronized := FALSE;
Active[slot].Duration    := T#0S;
Active[slot].Shelved     := FALSE;
Active[slot].ShelvedUntil:= DT#1970-01-01-00:00:00;
Active[slot].ShelfTimeSynchronized := FALSE;
_shelfMs[slot] := 0;
_comeMs[slot] := TIME_TO_DWORD(TIME());
NActive := NActive + 1;
_M_UpdateBlocking();
IF _sink <> 0 THEN
    _sink.OnEvent(Ev := Active[slot]);              // come notification (§8.3(d))
END_IF
_M_Raise := slot;
END_METHOD

// §8.3(c) — open an ERROR event straight from a first-out diagnostic (no re-authoring)
METHOD RaiseDiag : INT
VAR_INPUT
    D : ST_Diagnostic;
    ResetClass : E_ResetClass;
END_VAR
RaiseDiag := _M_Raise(Reason := D.ReasonCode, Text := D.Description,
                   Source := D.SourcePath, IoTag := D.IoTag, IoAddress := D.IoAddress,
                   Severity := D.Severity, Category := D.Category,
                   ResetClass := ResetClass);
END_METHOD

// §8.3(b) — condition re-established: AUTO_RESET closes with Duration;
// MANUAL_RESET stays blocking in WAIT_RESET until OperatorReset.
METHOD Gone : BOOL
VAR_INPUT
    Slot : INT;
END_VAR
Gone := FALSE;
IF (Slot < 1) OR (Slot > PL_Fraktal.MAX_ALARM_ACTIVE) THEN
    RETURN;
END_IF
IF Active[Slot].State <> E_AlarmState.ACTIVE THEN
    RETURN;
END_IF
Active[Slot].GoneAt   := F_Now();
Active[Slot].GoneTimeSynchronized := F_TimeSynchronized();
Active[Slot].Duration := DWORD_TO_TIME(TIME_TO_DWORD(TIME()) - _comeMs[Slot]);   // wrap-safe
IF Active[Slot].ResetClass = E_ResetClass.AUTO_RESET THEN
    _M_Close(Slot);
ELSE
    Active[Slot].State := E_AlarmState.WAIT_RESET;   // still blocking (§8.3(b))
END_IF
Gone := TRUE;
END_METHOD

// §8.3(b) — deliberate, release-gated operator action (§7.6/§14): closes a
// MANUAL_RESET event from WAIT_RESET *or* ACTIVE. NEVER self-invoked (§9.3 principle).
METHOD OperatorReset : BOOL
VAR
    i : INT;
END_VAR
OperatorReset := FALSE;
FOR i := 1 TO PL_Fraktal.MAX_ALARM_ACTIVE DO
    // Closing ONLY from WAIT_RESET made the reset a guaranteed no-op for exactly
    // the events that block restart. An ACTIVE MANUAL_RESET event sets Blocking,
    // so Start is refused; reaching WAIT_RESET needs the condition re-established,
    // and a condition such as "two-hand held during a stroke" can only be
    // re-established BY starting. Reset was the one action meant to break that
    // circle and it skipped the event entirely (real hard-lock on the press).
    // Closing a still-live cause is safe and self-correcting rather than a bypass:
    // its owner re-raises it on the next scan through the normal §8.3(c) capture,
    // and the interlock that withholds the output was never touched here.
    IF (Active[i].State = E_AlarmState.WAIT_RESET)
    OR ((Active[i].State = E_AlarmState.ACTIVE)
        AND (Active[i].ResetClass = E_ResetClass.MANUAL_RESET)) THEN
        IF Active[i].State = E_AlarmState.ACTIVE THEN
            // never received a Gone: stamp the come->reset span so the ring entry
            // still carries a Duration (§8.3(a)) instead of a zero.
            Active[i].GoneAt   := F_Now();
            Active[i].GoneTimeSynchronized := F_TimeSynchronized();
            Active[i].Duration := DWORD_TO_TIME(TIME_TO_DWORD(TIME()) - _comeMs[i]);
        END_IF
        Active[i].ResetAt := F_Now();
        Active[i].ResetTimeSynchronized := F_TimeSynchronized();
        _M_Close(i);
        OperatorReset := TRUE;
    END_IF
END_FOR
END_METHOD

METHOD SetSink : BOOL
VAR_INPUT
    Sink : I_EventSink;
END_VAR
_sink := Sink;
SetSink := TRUE;
END_METHOD

METHOD PRIVATE _M_Close
VAR_INPUT
    Slot : INT;
END_VAR
Active[Slot].State := E_AlarmState.CLOSED;
RingHead := (RingHead MOD PL_Fraktal.MAX_ALARM_RING) + 1;
Ring[RingHead] := Active[Slot];
Ring[RingHead].State := E_AlarmState.CLOSED;
NActive := NActive - 1;
_M_UpdateBlocking();
IF _sink <> 0 THEN
    _sink.OnEvent(Ev := Ring[RingHead]);            // close notification with Duration (§8.3(d))
END_IF
END_METHOD

METHOD PRIVATE _M_UpdateBlocking
VAR
    i : INT;
    b : BOOL;
END_VAR
b := FALSE;
FOR i := 1 TO PL_Fraktal.MAX_ALARM_ACTIVE DO
    IF (Active[i].ResetClass = E_ResetClass.MANUAL_RESET)
    AND (Active[i].State <> E_AlarmState.CLOSED) THEN
        b := TRUE;
        EXIT;
    END_IF
END_FOR
Blocking := b;
END_METHOD

// §8.9 compatibility helper for project reasons outside the generated registry.
// Standard reasons are generated and reject override; use RegisterMetaFull when
// an external reason needs non-default priority/category.
METHOD RegisterMeta : BOOL
VAR_INPUT
    Reason         : E_Reason;
    OperatorAction : STRING(255);
    Consequence    : STRING(255);
    Shelvable      : BOOL;
END_VAR
RegisterMeta := RegisterMetaFull(Reason := Reason,
    OperatorAction := OperatorAction, Consequence := Consequence,
    Priority := E_Severity.LOW, Category := E_Category.PROCESS,
    Shelvable := Shelvable);
END_METHOD

// §8.9 extension seam for application/type reasons outside the generated registry.
// Standard reasons reject here: their generated metadata is the single authority.
METHOD RegisterMetaFull : BOOL
VAR_INPUT
    Reason         : E_Reason;
    OperatorAction : STRING(255);
    Consequence    : STRING(255);
    Priority       : E_Severity;
    Category       : E_Category;
    Shelvable      : BOOL;
END_VAR
VAR
    i : INT;
    generated : ST_AlarmMeta;
END_VAR
RegisterMetaFull := FALSE;
IF F_ReasonMeta(Reason := Reason, Meta := generated) THEN
    RETURN;                              // generated standard metadata cannot drift
END_IF
IF (Reason = E_Reason.NONE) OR (OperatorAction = '') OR (Consequence = '') THEN
    RETURN;                              // complete actionable record required
END_IF
IF (TO_DINT(Priority) < TO_DINT(E_Severity.LOW))
OR (TO_DINT(Priority) > TO_DINT(E_Severity.HIGH))
OR (TO_DINT(Category) < TO_DINT(E_Category.PROCESS))
OR (TO_DINT(Category) > TO_DINT(E_Category.SYSTEM)) THEN
    RETURN;                              // non-strict transport enums still need bounds
END_IF
IF (Category = E_Category.SAFETY) AND Shelvable THEN
    RETURN;                              // §8.10: Safety is never shelvable
END_IF
FOR i := 1 TO MetaCount DO
    IF Meta[i].ReasonCode = Reason THEN
        Meta[i].OperatorAction := OperatorAction;
        Meta[i].Consequence := Consequence;
        Meta[i].Priority := Priority;
        Meta[i].Category := Category;
        Meta[i].Shelvable := Shelvable;
        RegisterMetaFull := TRUE;
        RETURN;
    END_IF
END_FOR
IF MetaCount >= PL_Fraktal.MAX_ALARM_META THEN
    RETURN;
END_IF
MetaCount := MetaCount + 1;
Meta[MetaCount].ReasonCode := Reason;
Meta[MetaCount].OperatorAction := OperatorAction;
Meta[MetaCount].Consequence := Consequence;
Meta[MetaCount].Priority := Priority;
Meta[MetaCount].Category := Category;
Meta[MetaCount].Shelvable := Shelvable;
RegisterMetaFull := TRUE;
END_METHOD

// §8.10 — may this active slot be shelved? SAFETY never; no meta record => no.
METHOD PROTECTED _M_Shelvable : BOOL
VAR_INPUT
    Slot : INT;
END_VAR
VAR
    i : INT;
    generated : ST_AlarmMeta;
END_VAR
_M_Shelvable := FALSE;
IF Slot < 1 OR Slot > PL_Fraktal.MAX_ALARM_ACTIVE THEN
    RETURN;
END_IF
IF Active[Slot].State = E_AlarmState.CLOSED THEN
    RETURN;
END_IF
IF Active[Slot].Category = E_Category.SAFETY THEN
    RETURN;                              // §8.10: safety never shelvable
END_IF
IF F_ReasonMeta(Reason := Active[Slot].ReasonCode, Meta := generated) THEN
    _M_Shelvable := generated.Shelvable;
    RETURN;
END_IF
FOR i := 1 TO MetaCount DO
    IF Meta[i].ReasonCode = Active[Slot].ReasonCode THEN
        _M_Shelvable := Meta[i].Shelvable;
        RETURN;
    END_IF
END_FOR
// no rationalization record => not shelvable (rationalize first, §8.10)
END_METHOD

// §8.10 — suppress ANNUNCIATION of an active alarm for DurationS seconds (capped).
// Control is untouched: Blocking, interlocks, release reports all still see it.
// Caller has already checked §7.7 ALARM_SHELVE; the shelf itself is logged here.
METHOD Shelve : BOOL
VAR_INPUT
    Slot      : INT;
    DurationS : UDINT;
END_VAR
VAR
    auditSlot : INT;
END_VAR
IF NOT _M_Shelvable(Slot := Slot) THEN
    Shelve := FALSE;
    RETURN;
END_IF
IF DurationS = 0 THEN
    Shelve := FALSE;                              // every shelf is time-bounded
    RETURN;
END_IF
IF DurationS > PL_Fraktal.MAX_SHELF_S THEN
    DurationS := PL_Fraktal.MAX_SHELF_S;         // §8.10 time-bounded
END_IF
Active[Slot].Shelved := TRUE;
Active[Slot].ShelvedUntil := DWORD_TO_DT(DT_TO_DWORD(F_Now()) + DurationS);
Active[Slot].ShelfTimeSynchronized := F_TimeSynchronized();
_shelfMs[Slot] := DurationS * 1000;
auditSlot := Raise(Reason := E_Reason.NONE,
    Text := 'std.audit.alarmShelved', Source := Active[Slot].SourcePath,
    Severity := E_Severity.LOW, Category := E_Category.SYSTEM, ResetClass := E_ResetClass.AUTO_RESET);
IF auditSlot > 0 THEN Gone(Slot := auditSlot); END_IF
Shelve := TRUE;
END_METHOD

// §8.10 — restore annunciation (operator or auto-expiry). Logged.
METHOD Unshelve : BOOL
VAR_INPUT
    Slot : INT;
END_VAR
VAR
    auditSlot : INT;
END_VAR
IF Slot < 1 OR Slot > PL_Fraktal.MAX_ALARM_ACTIVE THEN
    Unshelve := FALSE;
    RETURN;
END_IF
IF NOT Active[Slot].Shelved THEN
    Unshelve := FALSE;
    RETURN;
END_IF
Active[Slot].Shelved := FALSE;
_shelfMs[Slot] := 0;
auditSlot := Raise(Reason := E_Reason.NONE,
    Text := 'std.audit.alarmUnshelved', Source := Active[Slot].SourcePath,
    Severity := E_Severity.LOW, Category := E_Category.SYSTEM, ResetClass := E_ResetClass.AUTO_RESET);
IF auditSlot > 0 THEN Gone(Slot := auditSlot); END_IF
Unshelve := TRUE;
END_METHOD

// Resolve the HMI's stable alarm identity to exactly one live slot. Slot numbers
// are intentionally not persisted by the client because table reuse can retarget
// a stale request. Ambiguous duplicate identities fail closed.
METHOD FindActiveSlot : INT
VAR_INPUT
    SourcePath : STRING(255);
    Description : STRING(255);
END_VAR
VAR
    i : INT;
    found : INT;
END_VAR
found := 0;
IF (SourcePath = '') OR (Description = '') THEN
    FindActiveSlot := 0;
    RETURN;
END_IF
FOR i := 1 TO PL_Fraktal.MAX_ALARM_ACTIVE DO
    IF (Active[i].State <> E_AlarmState.CLOSED)
    AND (Active[i].SourcePath = SourcePath)
    AND (Active[i].Description = Description) THEN
        IF found <> 0 THEN
            FindActiveSlot := 0;                 // ambiguous identity: never guess
            RETURN;
        END_IF
        found := i;
    END_IF
END_FOR
FindActiveSlot := found;
END_METHOD

// §8.10 — auto-unshelve countdown (owning Unit ticks this each scan).
METHOD Cyclic : BOOL
VAR
    currentTime : TIME;
    deltaMs     : UDINT;
    i   : INT;
END_VAR
currentTime := TIME();                 // monotonic duration clock
IF _cycLast = T#0S THEN
    _cycLast := currentTime;
    Cyclic := TRUE;
    RETURN;
END_IF
deltaMs := TIME_TO_UDINT(currentTime) - TIME_TO_UDINT(_cycLast);
_cycLast := currentTime;
FOR i := 1 TO PL_Fraktal.MAX_ALARM_ACTIVE DO
    IF Active[i].Shelved AND _shelfMs[i] > 0 THEN
        IF _shelfMs[i] > deltaMs THEN
            _shelfMs[i] := _shelfMs[i] - deltaMs;
        ELSE
            _shelfMs[i] := 0;
            Unshelve(Slot := i);                 // §8.10 auto-expire (logged by Unshelve)
        END_IF
    END_IF
END_FOR
Cyclic := TRUE;
END_METHOD

END_FUNCTION_BLOCK

// ---- Platform/F_EngUnitSymbol.TcPOU
// Core §3.10.2 - the ASCII symbol for a unit code, published as the entry's
// legacy Unit text so a client that predates UnitCode still shows a unit. It is
// DERIVED from the code, never a second source: the code is the contract, and a
// current HMI shows its own translated symbol (std.unit.<name>) instead.
FUNCTION F_EngUnitSymbol : STRING(16)
VAR_INPUT
    Unit : E_EngUnit;
END_VAR

CASE Unit OF
    E_EngUnit.NONE:                          F_EngUnitSymbol := '';
    E_EngUnit.MILLISECOND:                   F_EngUnitSymbol := 'ms';
    E_EngUnit.SECOND:                        F_EngUnitSymbol := 's';
    E_EngUnit.MINUTE:                        F_EngUnitSymbol := 'min';
    E_EngUnit.HOUR:                          F_EngUnitSymbol := 'h';
    E_EngUnit.MICROMETER:                    F_EngUnitSymbol := 'um';
    E_EngUnit.MILLIMETER:                    F_EngUnitSymbol := 'mm';
    E_EngUnit.METER:                         F_EngUnitSymbol := 'm';
    E_EngUnit.DEGREE:                        F_EngUnitSymbol := 'deg';
    E_EngUnit.MILLIMETER_PER_SECOND:         F_EngUnitSymbol := 'mm/s';
    E_EngUnit.METER_PER_MINUTE:              F_EngUnitSymbol := 'm/min';
    E_EngUnit.DEGREE_PER_SECOND:             F_EngUnitSymbol := 'deg/s';
    E_EngUnit.MILLIMETER_PER_SECOND_SQUARED: F_EngUnitSymbol := 'mm/s2';
    E_EngUnit.BAR:                           F_EngUnitSymbol := 'bar';
    E_EngUnit.KILOPASCAL:                    F_EngUnitSymbol := 'kPa';
    E_EngUnit.NEWTON:                        F_EngUnitSymbol := 'N';
    E_EngUnit.KILONEWTON:                    F_EngUnitSymbol := 'kN';
    E_EngUnit.NEWTON_METER:                  F_EngUnitSymbol := 'Nm';
    E_EngUnit.GRAM:                          F_EngUnitSymbol := 'g';
    E_EngUnit.KILOGRAM:                      F_EngUnitSymbol := 'kg';
    E_EngUnit.DEGREE_CELSIUS:                F_EngUnitSymbol := 'degC';
    E_EngUnit.PERCENT:                       F_EngUnitSymbol := '%';
    E_EngUnit.REVOLUTION_PER_MINUTE:         F_EngUnitSymbol := 'rpm';
    E_EngUnit.HERTZ:                         F_EngUnitSymbol := 'Hz';
    E_EngUnit.VOLT:                          F_EngUnitSymbol := 'V';
    E_EngUnit.AMPERE:                        F_EngUnitSymbol := 'A';
    E_EngUnit.WATT:                          F_EngUnitSymbol := 'W';
    E_EngUnit.KILOWATT:                      F_EngUnitSymbol := 'kW';
    E_EngUnit.LITER:                         F_EngUnitSymbol := 'l';
    E_EngUnit.LITER_PER_MINUTE:              F_EngUnitSymbol := 'l/min';
    E_EngUnit.PIECE:                         F_EngUnitSymbol := 'pcs';
    E_EngUnit.PIECE_PER_MINUTE:              F_EngUnitSymbol := 'pcs/min';
    E_EngUnit.PIECE_PER_HOUR:                F_EngUnitSymbol := 'pcs/h';
ELSE
    F_EngUnitSymbol := '';                   // an unknown code shows no unit
END_CASE

END_FUNCTION

